KUKA KRL program: Jacob_final_print.src

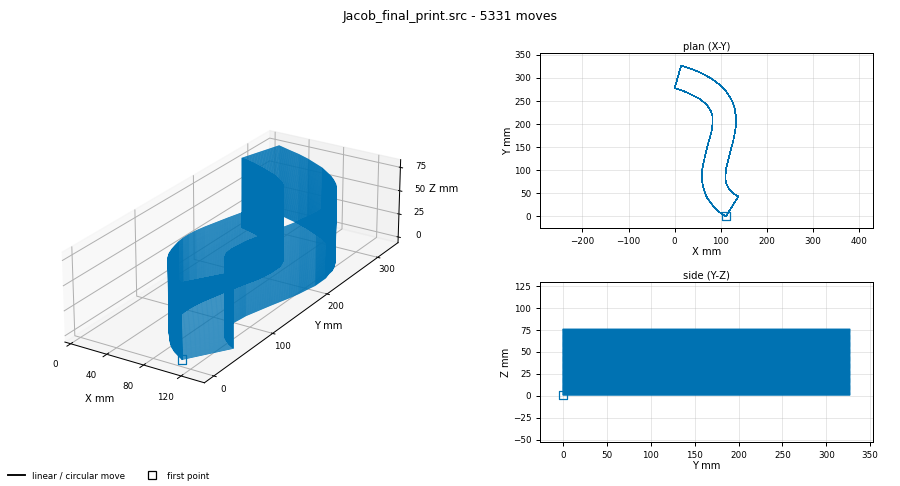
[picture p0: tool path of Jacob_final_print.src, 5331 of 5334 moves have a stored position in this frame; points joined in program order, loops and branches not executed]
&ACCESS RVP
&REL 25
DEF Jacob_final_print()

;FOLD INI
  ;FOLD BASISTECH INI
    GLOBAL INTERRUPT DECL 3 WHEN $STOPMESS==TRUE DO IR_STOPM ( )
    INTERRUPT ON 3
    BAS (#INITMOV,0 )
  ;ENDFOLD (BASISTECH INI)
  ;FOLD USER INI
    ;Make your modifications here

  ;ENDFOLD (USER INI)
;ENDFOLD (INI)

;FOLD PTP HOME  Vel= 100 % DEFAULT;%{PE}%R 5.4.37,%MKUKATPBASIS,%CMOVE,%VPTP,%P 1:PTP, 2:HOME, 3:, 5:100, 7:DEFAULT
$BWDSTART=FALSE
PDAT_ACT=PDEFAULT
FDAT_ACT=FHOME
BAS(#PTP_PARAMS,100)
$H_POS=XHOME
PTP XHOME
;ENDFOLD

$VEL_AXIS[1]=20
$VEL_AXIS[2]=20
$VEL_AXIS[3]=20
$VEL_AXIS[4]=20
$VEL_AXIS[5]=20
$VEL_AXIS[6]=20

$vel.cp= 0.30
$apo.cvel= 95

PTP {A1 0, A2 -90, A3 90, A4 0, A5 0, A6 0}

PTP {Z 450, S 110}

LIN {X 111, Y 0, Z 1} c_vel
$OUT[4] = TRUE
LIN {X 111, Y 0, Z 1} c_vel
LIN {X 106, Y 3, Z 1} c_vel
LIN {X 97, Y 9, Z 1} c_vel
LIN {X 89, Y 16, Z 1} c_vel
LIN {X 83, Y 23, Z 1} c_vel
LIN {X 77, Y 31, Z 1} c_vel
LIN {X 71, Y 39, Z 1} c_vel
LIN {X 67, Y 47, Z 1} c_vel
LIN {X 64, Y 56, Z 1} c_vel
LIN {X 62, Y 64, Z 1} c_vel
LIN {X 60, Y 73, Z 1} c_vel
LIN {X 59, Y 82, Z 1} c_vel
LIN {X 59, Y 82, Z 1} c_vel
LIN {X 59, Y 92, Z 1} c_vel
LIN {X 60, Y 103, Z 1} c_vel
LIN {X 62, Y 114, Z 1} c_vel
LIN {X 65, Y 127, Z 1} c_vel
LIN {X 69, Y 144, Z 1} c_vel
LIN {X 74, Y 163, Z 1} c_vel
LIN {X 79, Y 180, Z 1} c_vel
LIN {X 81, Y 191, Z 1} c_vel
LIN {X 82, Y 201, Z 1} c_vel
LIN {X 82, Y 209, Z 1} c_vel
LIN {X 82, Y 217, Z 1} c_vel
LIN {X 80, Y 223, Z 1} c_vel
LIN {X 78, Y 229, Z 1} c_vel
LIN {X 75, Y 234, Z 1} c_vel
LIN {X 71, Y 240, Z 1} c_vel
LIN {X 66, Y 245, Z 1} c_vel
LIN {X 60, Y 250, Z 1} c_vel
LIN {X 52, Y 256, Z 1} c_vel
LIN {X 42, Y 261, Z 1} c_vel
LIN {X 30, Y 267, Z 1} c_vel
LIN {X 16, Y 273, Z 1} c_vel
LIN {X 0, Y 278, Z 1} c_vel
LIN {X 14, Y 327, Z 1} c_vel
LIN {X 28, Y 322, Z 1} c_vel
LIN {X 43, Y 317, Z 1} c_vel
LIN {X 57, Y 311, Z 1} c_vel
LIN {X 70, Y 304, Z 1} c_vel
LIN {X 81, Y 298, Z 1} c_vel
LIN {X 90, Y 291, Z 1} c_vel
LIN {X 99, Y 284, Z 1} c_vel
LIN {X 106, Y 277, Z 1} c_vel
LIN {X 113, Y 269, Z 1} c_vel
LIN {X 118, Y 261, Z 1} c_vel
LIN {X 123, Y 253, Z 1} c_vel
LIN {X 127, Y 244, Z 1} c_vel
LIN {X 130, Y 235, Z 1} c_vel
LIN {X 131, Y 226, Z 1} c_vel
LIN {X 133, Y 217, Z 1} c_vel
LIN {X 133, Y 207, Z 1} c_vel
LIN {X 133, Y 197, Z 1} c_vel
LIN {X 131, Y 186, Z 1} c_vel
LIN {X 129, Y 173, Z 1} c_vel
LIN {X 126, Y 160, Z 1} c_vel
LIN {X 120, Y 138, Z 1} c_vel
LIN {X 115, Y 118, Z 1} c_vel
LIN {X 112, Y 106, Z 1} c_vel
LIN {X 111, Y 96, Z 1} c_vel
LIN {X 110, Y 88, Z 1} c_vel
LIN {X 110, Y 81, Z 1} c_vel
LIN {X 111, Y 74, Z 1} c_vel
LIN {X 113, Y 69, Z 1} c_vel
LIN {X 116, Y 63, Z 1} c_vel
LIN {X 119, Y 58, Z 1} c_vel
LIN {X 124, Y 53, Z 1} c_vel
LIN {X 130, Y 48, Z 1} c_vel
LIN {X 138, Y 43, Z 1} c_vel
LIN {X 111, Y 0, Z 1} c_vel
$OUT[4] = FALSE
WAIT SEC 10.0
LIN {X 111, Y 0, Z 2} c_vel
$OUT[4] = TRUE
LIN {X 111, Y 0, Z 2} c_vel
LIN {X 106, Y 3, Z 2} c_vel
LIN {X 97, Y 9, Z 2} c_vel
LIN {X 89, Y 16, Z 2} c_vel
LIN {X 83, Y 23, Z 2} c_vel
LIN {X 77, Y 31, Z 2} c_vel
LIN {X 71, Y 39, Z 2} c_vel
LIN {X 67, Y 47, Z 2} c_vel
LIN {X 64, Y 56, Z 2} c_vel
LIN {X 62, Y 64, Z 2} c_vel
LIN {X 60, Y 73, Z 2} c_vel
LIN {X 59, Y 82, Z 2} c_vel
LIN {X 59, Y 83, Z 2} c_vel
LIN {X 59, Y 92, Z 2} c_vel
LIN {X 60, Y 103, Z 2} c_vel
LIN {X 62, Y 114, Z 2} c_vel
LIN {X 65, Y 127, Z 2} c_vel
LIN {X 69, Y 144, Z 2} c_vel
LIN {X 74, Y 163, Z 2} c_vel
LIN {X 79, Y 180, Z 2} c_vel
LIN {X 81, Y 191, Z 2} c_vel
LIN {X 82, Y 201, Z 2} c_vel
LIN {X 82, Y 209, Z 2} c_vel
LIN {X 82, Y 217, Z 2} c_vel
LIN {X 80, Y 223, Z 2} c_vel
LIN {X 78, Y 229, Z 2} c_vel
LIN {X 75, Y 234, Z 2} c_vel
LIN {X 71, Y 240, Z 2} c_vel
LIN {X 66, Y 245, Z 2} c_vel
LIN {X 60, Y 250, Z 2} c_vel
LIN {X 52, Y 256, Z 2} c_vel
LIN {X 42, Y 261, Z 2} c_vel
LIN {X 30, Y 267, Z 2} c_vel
LIN {X 16, Y 273, Z 2} c_vel
LIN {X 0, Y 278, Z 2} c_vel
LIN {X 14, Y 327, Z 2} c_vel
LIN {X 28, Y 322, Z 2} c_vel
LIN {X 43, Y 317, Z 2} c_vel
LIN {X 57, Y 311, Z 2} c_vel
LIN {X 70, Y 304, Z 2} c_vel
LIN {X 81, Y 298, Z 2} c_vel
LIN {X 90, Y 291, Z 2} c_vel
LIN {X 99, Y 284, Z 2} c_vel
LIN {X 106, Y 277, Z 2} c_vel
LIN {X 113, Y 269, Z 2} c_vel
LIN {X 118, Y 261, Z 2} c_vel
LIN {X 123, Y 253, Z 2} c_vel
LIN {X 127, Y 244, Z 2} c_vel
LIN {X 130, Y 235, Z 2} c_vel
LIN {X 131, Y 226, Z 2} c_vel
LIN {X 133, Y 217, Z 2} c_vel
LIN {X 133, Y 207, Z 2} c_vel
LIN {X 133, Y 197, Z 2} c_vel
LIN {X 131, Y 186, Z 2} c_vel
LIN {X 129, Y 173, Z 2} c_vel
LIN {X 126, Y 160, Z 2} c_vel
LIN {X 120, Y 138, Z 2} c_vel
LIN {X 115, Y 118, Z 2} c_vel
LIN {X 112, Y 106, Z 2} c_vel
LIN {X 111, Y 96, Z 2} c_vel
LIN {X 110, Y 88, Z 2} c_vel
LIN {X 110, Y 81, Z 2} c_vel
LIN {X 111, Y 74, Z 2} c_vel
LIN {X 113, Y 69, Z 2} c_vel
LIN {X 116, Y 63, Z 2} c_vel
LIN {X 119, Y 58, Z 2} c_vel
LIN {X 124, Y 53, Z 2} c_vel
LIN {X 130, Y 48, Z 2} c_vel
LIN {X 138, Y 43, Z 2} c_vel
LIN {X 111, Y 0, Z 2} c_vel
$OUT[4] = FALSE
WAIT SEC 10.0
LIN {X 111, Y 0, Z 3} c_vel
$OUT[4] = TRUE
LIN {X 111, Y 0, Z 3} c_vel
LIN {X 106, Y 3, Z 3} c_vel
LIN {X 97, Y 9, Z 3} c_vel
LIN {X 89, Y 16, Z 3} c_vel
LIN {X 83, Y 23, Z 3} c_vel
LIN {X 77, Y 31, Z 3} c_vel
LIN {X 71, Y 39, Z 3} c_vel
LIN {X 67, Y 47, Z 3} c_vel
LIN {X 64, Y 56, Z 3} c_vel
LIN {X 62, Y 64, Z 3} c_vel
LIN {X 60, Y 73, Z 3} c_vel
LIN {X 59, Y 82, Z 3} c_vel
LIN {X 59, Y 83, Z 3} c_vel
LIN {X 59, Y 92, Z 3} c_vel
LIN {X 60, Y 103, Z 3} c_vel
LIN {X 62, Y 114, Z 3} c_vel
LIN {X 65, Y 127, Z 3} c_vel
LIN {X 69, Y 144, Z 3} c_vel
LIN {X 74, Y 163, Z 3} c_vel
LIN {X 79, Y 180, Z 3} c_vel
LIN {X 81, Y 191, Z 3} c_vel
LIN {X 82, Y 201, Z 3} c_vel
LIN {X 82, Y 209, Z 3} c_vel
LIN {X 82, Y 217, Z 3} c_vel
LIN {X 80, Y 223, Z 3} c_vel
LIN {X 78, Y 229, Z 3} c_vel
LIN {X 75, Y 234, Z 3} c_vel
LIN {X 71, Y 240, Z 3} c_vel
LIN {X 66, Y 245, Z 3} c_vel
LIN {X 60, Y 250, Z 3} c_vel
LIN {X 52, Y 256, Z 3} c_vel
LIN {X 42, Y 261, Z 3} c_vel
LIN {X 30, Y 267, Z 3} c_vel
LIN {X 16, Y 273, Z 3} c_vel
LIN {X 0, Y 278, Z 3} c_vel
LIN {X 14, Y 327, Z 3} c_vel
LIN {X 28, Y 322, Z 3} c_vel
LIN {X 43, Y 317, Z 3} c_vel
LIN {X 57, Y 311, Z 3} c_vel
LIN {X 70, Y 304, Z 3} c_vel
LIN {X 81, Y 298, Z 3} c_vel
LIN {X 90, Y 291, Z 3} c_vel
LIN {X 99, Y 284, Z 3} c_vel
LIN {X 106, Y 277, Z 3} c_vel
LIN {X 113, Y 269, Z 3} c_vel
LIN {X 118, Y 261, Z 3} c_vel
LIN {X 123, Y 253, Z 3} c_vel
LIN {X 127, Y 244, Z 3} c_vel
LIN {X 130, Y 235, Z 3} c_vel
LIN {X 131, Y 226, Z 3} c_vel
LIN {X 133, Y 217, Z 3} c_vel
LIN {X 133, Y 207, Z 3} c_vel
LIN {X 133, Y 197, Z 3} c_vel
LIN {X 131, Y 186, Z 3} c_vel
LIN {X 129, Y 173, Z 3} c_vel
LIN {X 126, Y 160, Z 3} c_vel
LIN {X 120, Y 138, Z 3} c_vel
LIN {X 115, Y 118, Z 3} c_vel
LIN {X 112, Y 106, Z 3} c_vel
LIN {X 111, Y 96, Z 3} c_vel
LIN {X 110, Y 88, Z 3} c_vel
LIN {X 110, Y 81, Z 3} c_vel
LIN {X 111, Y 74, Z 3} c_vel
LIN {X 113, Y 69, Z 3} c_vel
LIN {X 116, Y 63, Z 3} c_vel
LIN {X 119, Y 58, Z 3} c_vel
LIN {X 124, Y 53, Z 3} c_vel
LIN {X 130, Y 48, Z 3} c_vel
LIN {X 138, Y 43, Z 3} c_vel
LIN {X 111, Y 0, Z 3} c_vel
$OUT[4] = FALSE
WAIT SEC 10.0
LIN {X 111, Y 0, Z 4} c_vel
$OUT[4] = TRUE
LIN {X 111, Y 0, Z 4} c_vel
LIN {X 106, Y 3, Z 4} c_vel
LIN {X 97, Y 9, Z 4} c_vel
LIN {X 89, Y 16, Z 4} c_vel
LIN {X 83, Y 23, Z 4} c_vel
LIN {X 77, Y 31, Z 4} c_vel
LIN {X 71, Y 39, Z 4} c_vel
LIN {X 67, Y 47, Z 4} c_vel
LIN {X 64, Y 56, Z 4} c_vel
LIN {X 62, Y 64, Z 4} c_vel
LIN {X 60, Y 73, Z 4} c_vel
LIN {X 59, Y 82, Z 4} c_vel
LIN {X 59, Y 83, Z 4} c_vel
LIN {X 59, Y 92, Z 4} c_vel
LIN {X 60, Y 103, Z 4} c_vel
LIN {X 62, Y 114, Z 4} c_vel
LIN {X 65, Y 127, Z 4} c_vel
LIN {X 69, Y 144, Z 4} c_vel
LIN {X 74, Y 163, Z 4} c_vel
LIN {X 79, Y 180, Z 4} c_vel
LIN {X 81, Y 191, Z 4} c_vel
LIN {X 82, Y 201, Z 4} c_vel
LIN {X 82, Y 209, Z 4} c_vel
LIN {X 82, Y 217, Z 4} c_vel
LIN {X 80, Y 223, Z 4} c_vel
LIN {X 78, Y 229, Z 4} c_vel
LIN {X 75, Y 234, Z 4} c_vel
LIN {X 71, Y 240, Z 4} c_vel
LIN {X 66, Y 245, Z 4} c_vel
LIN {X 60, Y 250, Z 4} c_vel
LIN {X 52, Y 256, Z 4} c_vel
LIN {X 42, Y 261, Z 4} c_vel
LIN {X 30, Y 267, Z 4} c_vel
LIN {X 16, Y 273, Z 4} c_vel
LIN {X 0, Y 278, Z 4} c_vel
LIN {X 14, Y 327, Z 4} c_vel
LIN {X 28, Y 322, Z 4} c_vel
LIN {X 43, Y 317, Z 4} c_vel
LIN {X 57, Y 311, Z 4} c_vel
LIN {X 70, Y 304, Z 4} c_vel
LIN {X 81, Y 298, Z 4} c_vel
LIN {X 90, Y 291, Z 4} c_vel
LIN {X 99, Y 284, Z 4} c_vel
LIN {X 106, Y 277, Z 4} c_vel
LIN {X 113, Y 269, Z 4} c_vel
LIN {X 118, Y 261, Z 4} c_vel
LIN {X 123, Y 253, Z 4} c_vel
LIN {X 127, Y 244, Z 4} c_vel
LIN {X 130, Y 235, Z 4} c_vel
LIN {X 131, Y 226, Z 4} c_vel
LIN {X 133, Y 217, Z 4} c_vel
LIN {X 133, Y 207, Z 4} c_vel
LIN {X 133, Y 197, Z 4} c_vel
LIN {X 131, Y 186, Z 4} c_vel
LIN {X 129, Y 173, Z 4} c_vel
LIN {X 126, Y 160, Z 4} c_vel
LIN {X 120, Y 138, Z 4} c_vel
LIN {X 115, Y 118, Z 4} c_vel
LIN {X 112, Y 106, Z 4} c_vel
LIN {X 111, Y 96, Z 4} c_vel
LIN {X 110, Y 88, Z 4} c_vel
LIN {X 110, Y 81, Z 4} c_vel
LIN {X 111, Y 74, Z 4} c_vel
LIN {X 113, Y 69, Z 4} c_vel
LIN {X 116, Y 63, Z 4} c_vel
LIN {X 119, Y 58, Z 4} c_vel
LIN {X 124, Y 53, Z 4} c_vel
LIN {X 130, Y 48, Z 4} c_vel
LIN {X 138, Y 43, Z 4} c_vel
LIN {X 111, Y 0, Z 4} c_vel
$OUT[4] = FALSE
WAIT SEC 10.0
LIN {X 111, Y 0, Z 5} c_vel
$OUT[4] = TRUE
LIN {X 111, Y 0, Z 5} c_vel
LIN {X 106, Y 3, Z 5} c_vel
LIN {X 97, Y 9, Z 5} c_vel
LIN {X 89, Y 16, Z 5} c_vel
LIN {X 83, Y 23, Z 5} c_vel
LIN {X 77, Y 31, Z 5} c_vel
LIN {X 71, Y 39, Z 5} c_vel
LIN {X 67, Y 47, Z 5} c_vel
LIN {X 64, Y 56, Z 5} c_vel
LIN {X 62, Y 64, Z 5} c_vel
LIN {X 60, Y 73, Z 5} c_vel
LIN {X 59, Y 82, Z 5} c_vel
LIN {X 59, Y 83, Z 5} c_vel
LIN {X 59, Y 92, Z 5} c_vel
LIN {X 60, Y 103, Z 5} c_vel
LIN {X 62, Y 114, Z 5} c_vel
LIN {X 65, Y 127, Z 5} c_vel
LIN {X 69, Y 144, Z 5} c_vel
LIN {X 74, Y 163, Z 5} c_vel
LIN {X 79, Y 180, Z 5} c_vel
LIN {X 81, Y 191, Z 5} c_vel
LIN {X 82, Y 201, Z 5} c_vel
LIN {X 82, Y 209, Z 5} c_vel
LIN {X 82, Y 217, Z 5} c_vel
LIN {X 80, Y 223, Z 5} c_vel
LIN {X 78, Y 229, Z 5} c_vel
LIN {X 75, Y 234, Z 5} c_vel
LIN {X 71, Y 240, Z 5} c_vel
LIN {X 66, Y 245, Z 5} c_vel
LIN {X 60, Y 250, Z 5} c_vel
LIN {X 52, Y 256, Z 5} c_vel
LIN {X 42, Y 261, Z 5} c_vel
LIN {X 30, Y 267, Z 5} c_vel
LIN {X 16, Y 273, Z 5} c_vel
LIN {X 0, Y 278, Z 5} c_vel
LIN {X 14, Y 327, Z 5} c_vel
LIN {X 28, Y 322, Z 5} c_vel
LIN {X 43, Y 317, Z 5} c_vel
LIN {X 57, Y 311, Z 5} c_vel
LIN {X 70, Y 304, Z 5} c_vel
LIN {X 81, Y 298, Z 5} c_vel
LIN {X 90, Y 291, Z 5} c_vel
LIN {X 99, Y 284, Z 5} c_vel
LIN {X 106, Y 277, Z 5} c_vel
LIN {X 113, Y 269, Z 5} c_vel
LIN {X 118, Y 261, Z 5} c_vel
LIN {X 123, Y 253, Z 5} c_vel
LIN {X 127, Y 244, Z 5} c_vel
LIN {X 130, Y 235, Z 5} c_vel
LIN {X 131, Y 226, Z 5} c_vel
LIN {X 133, Y 217, Z 5} c_vel
LIN {X 133, Y 207, Z 5} c_vel
LIN {X 133, Y 197, Z 5} c_vel
LIN {X 131, Y 186, Z 5} c_vel
LIN {X 129, Y 173, Z 5} c_vel
LIN {X 126, Y 160, Z 5} c_vel
LIN {X 120, Y 138, Z 5} c_vel
LIN {X 115, Y 118, Z 5} c_vel
LIN {X 112, Y 106, Z 5} c_vel
LIN {X 111, Y 96, Z 5} c_vel
LIN {X 110, Y 88, Z 5} c_vel
LIN {X 110, Y 81, Z 5} c_vel
LIN {X 111, Y 74, Z 5} c_vel
LIN {X 113, Y 69, Z 5} c_vel
LIN {X 116, Y 63, Z 5} c_vel
LIN {X 119, Y 58, Z 5} c_vel
LIN {X 124, Y 53, Z 5} c_vel
LIN {X 130, Y 48, Z 5} c_vel
LIN {X 138, Y 43, Z 5} c_vel
LIN {X 111, Y 0, Z 5} c_vel
$OUT[4] = FALSE
WAIT SEC 10.0
LIN {X 111, Y 0, Z 6} c_vel
$OUT[4] = TRUE
LIN {X 111, Y 0, Z 6} c_vel
LIN {X 106, Y 3, Z 6} c_vel
LIN {X 97, Y 9, Z 6} c_vel
LIN {X 89, Y 16, Z 6} c_vel
LIN {X 83, Y 23, Z 6} c_vel
LIN {X 77, Y 31, Z 6} c_vel
LIN {X 71, Y 39, Z 6} c_vel
LIN {X 67, Y 47, Z 6} c_vel
LIN {X 64, Y 56, Z 6} c_vel
LIN {X 62, Y 64, Z 6} c_vel
LIN {X 60, Y 73, Z 6} c_vel
LIN {X 59, Y 82, Z 6} c_vel
LIN {X 59, Y 83, Z 6} c_vel
LIN {X 59, Y 92, Z 6} c_vel
LIN {X 60, Y 103, Z 6} c_vel
LIN {X 62, Y 114, Z 6} c_vel
LIN {X 65, Y 127, Z 6} c_vel
LIN {X 69, Y 144, Z 6} c_vel
LIN {X 74, Y 163, Z 6} c_vel
LIN {X 79, Y 180, Z 6} c_vel
LIN {X 81, Y 191, Z 6} c_vel
LIN {X 82, Y 201, Z 6} c_vel
LIN {X 82, Y 209, Z 6} c_vel
LIN {X 82, Y 217, Z 6} c_vel
LIN {X 80, Y 223, Z 6} c_vel
LIN {X 78, Y 229, Z 6} c_vel
LIN {X 75, Y 234, Z 6} c_vel
LIN {X 71, Y 240, Z 6} c_vel
LIN {X 66, Y 245, Z 6} c_vel
LIN {X 60, Y 250, Z 6} c_vel
LIN {X 52, Y 256, Z 6} c_vel
LIN {X 42, Y 261, Z 6} c_vel
LIN {X 30, Y 267, Z 6} c_vel
LIN {X 16, Y 273, Z 6} c_vel
LIN {X 0, Y 278, Z 6} c_vel
LIN {X 14, Y 327, Z 6} c_vel
LIN {X 28, Y 322, Z 6} c_vel
LIN {X 43, Y 317, Z 6} c_vel
LIN {X 57, Y 311, Z 6} c_vel
LIN {X 70, Y 304, Z 6} c_vel
LIN {X 81, Y 298, Z 6} c_vel
LIN {X 90, Y 291, Z 6} c_vel
LIN {X 99, Y 284, Z 6} c_vel
LIN {X 106, Y 277, Z 6} c_vel
LIN {X 113, Y 269, Z 6} c_vel
LIN {X 118, Y 261, Z 6} c_vel
LIN {X 123, Y 253, Z 6} c_vel
LIN {X 127, Y 244, Z 6} c_vel
LIN {X 130, Y 235, Z 6} c_vel
LIN {X 131, Y 226, Z 6} c_vel
LIN {X 133, Y 217, Z 6} c_vel
LIN {X 133, Y 207, Z 6} c_vel
LIN {X 133, Y 197, Z 6} c_vel
LIN {X 131, Y 186, Z 6} c_vel
LIN {X 129, Y 173, Z 6} c_vel
LIN {X 126, Y 160, Z 6} c_vel
LIN {X 120, Y 138, Z 6} c_vel
LIN {X 115, Y 118, Z 6} c_vel
LIN {X 112, Y 106, Z 6} c_vel
LIN {X 111, Y 96, Z 6} c_vel
LIN {X 110, Y 88, Z 6} c_vel
LIN {X 110, Y 81, Z 6} c_vel
LIN {X 111, Y 74, Z 6} c_vel
LIN {X 113, Y 69, Z 6} c_vel
LIN {X 116, Y 63, Z 6} c_vel
LIN {X 119, Y 58, Z 6} c_vel
LIN {X 124, Y 53, Z 6} c_vel
LIN {X 130, Y 48, Z 6} c_vel
LIN {X 138, Y 43, Z 6} c_vel
LIN {X 111, Y 0, Z 6} c_vel
$OUT[4] = FALSE
WAIT SEC 10.0
LIN {X 111, Y 0, Z 7} c_vel
$OUT[4] = TRUE
LIN {X 111, Y 0, Z 7} c_vel
LIN {X 106, Y 3, Z 7} c_vel
LIN {X 97, Y 9, Z 7} c_vel
LIN {X 89, Y 16, Z 7} c_vel
LIN {X 83, Y 23, Z 7} c_vel
LIN {X 77, Y 31, Z 7} c_vel
LIN {X 71, Y 39, Z 7} c_vel
LIN {X 67, Y 47, Z 7} c_vel
LIN {X 64, Y 56, Z 7} c_vel
LIN {X 62, Y 64, Z 7} c_vel
LIN {X 60, Y 73, Z 7} c_vel
LIN {X 59, Y 82, Z 7} c_vel
LIN {X 59, Y 92, Z 7} c_vel
LIN {X 60, Y 103, Z 7} c_vel
LIN {X 62, Y 114, Z 7} c_vel
LIN {X 65, Y 127, Z 7} c_vel
LIN {X 69, Y 144, Z 7} c_vel
LIN {X 74, Y 163, Z 7} c_vel
LIN {X 79, Y 180, Z 7} c_vel
LIN {X 81, Y 191, Z 7} c_vel
LIN {X 82, Y 201, Z 7} c_vel
LIN {X 82, Y 209, Z 7} c_vel
LIN {X 82, Y 217, Z 7} c_vel
LIN {X 80, Y 223, Z 7} c_vel
LIN {X 78, Y 229, Z 7} c_vel
LIN {X 75, Y 234, Z 7} c_vel
LIN {X 71, Y 240, Z 7} c_vel
LIN {X 66, Y 245, Z 7} c_vel
LIN {X 60, Y 250, Z 7} c_vel
LIN {X 52, Y 256, Z 7} c_vel
LIN {X 42, Y 261, Z 7} c_vel
LIN {X 30, Y 267, Z 7} c_vel
LIN {X 16, Y 273, Z 7} c_vel
LIN {X 0, Y 278, Z 7} c_vel
LIN {X 14, Y 327, Z 7} c_vel
LIN {X 28, Y 322, Z 7} c_vel
LIN {X 43, Y 317, Z 7} c_vel
LIN {X 57, Y 311, Z 7} c_vel
LIN {X 70, Y 304, Z 7} c_vel
LIN {X 81, Y 298, Z 7} c_vel
LIN {X 90, Y 291, Z 7} c_vel
LIN {X 99, Y 284, Z 7} c_vel
LIN {X 106, Y 277, Z 7} c_vel
LIN {X 113, Y 269, Z 7} c_vel
LIN {X 118, Y 261, Z 7} c_vel
LIN {X 123, Y 253, Z 7} c_vel
LIN {X 127, Y 244, Z 7} c_vel
LIN {X 130, Y 235, Z 7} c_vel
LIN {X 131, Y 226, Z 7} c_vel
LIN {X 133, Y 217, Z 7} c_vel
LIN {X 133, Y 207, Z 7} c_vel
LIN {X 133, Y 197, Z 7} c_vel
LIN {X 131, Y 186, Z 7} c_vel
LIN {X 129, Y 173, Z 7} c_vel
LIN {X 126, Y 160, Z 7} c_vel
LIN {X 120, Y 138, Z 7} c_vel
LIN {X 115, Y 118, Z 7} c_vel
LIN {X 112, Y 106, Z 7} c_vel
LIN {X 111, Y 96, Z 7} c_vel
LIN {X 110, Y 88, Z 7} c_vel
LIN {X 110, Y 81, Z 7} c_vel
LIN {X 111, Y 74, Z 7} c_vel
LIN {X 113, Y 69, Z 7} c_vel
LIN {X 116, Y 63, Z 7} c_vel
LIN {X 119, Y 58, Z 7} c_vel
LIN {X 124, Y 53, Z 7} c_vel
LIN {X 130, Y 48, Z 7} c_vel
LIN {X 138, Y 43, Z 7} c_vel
LIN {X 111, Y 0, Z 7} c_vel
$OUT[4] = FALSE
WAIT SEC 10.0
LIN {X 111, Y 0, Z 8} c_vel
$OUT[4] = TRUE
LIN {X 111, Y 0, Z 8} c_vel
LIN {X 106, Y 3, Z 8} c_vel
LIN {X 97, Y 9, Z 8} c_vel
LIN {X 89, Y 16, Z 8} c_vel
LIN {X 83, Y 23, Z 8} c_vel
LIN {X 77, Y 31, Z 8} c_vel
LIN {X 71, Y 39, Z 8} c_vel
LIN {X 67, Y 47, Z 8} c_vel
LIN {X 64, Y 56, Z 8} c_vel
LIN {X 62, Y 64, Z 8} c_vel
LIN {X 60, Y 73, Z 8} c_vel
LIN {X 59, Y 82, Z 8} c_vel
LIN {X 59, Y 92, Z 8} c_vel
LIN {X 60, Y 103, Z 8} c_vel
LIN {X 62, Y 114, Z 8} c_vel
LIN {X 65, Y 127, Z 8} c_vel
LIN {X 69, Y 144, Z 8} c_vel
LIN {X 74, Y 163, Z 8} c_vel
LIN {X 79, Y 180, Z 8} c_vel
LIN {X 81, Y 191, Z 8} c_vel
LIN {X 82, Y 201, Z 8} c_vel
LIN {X 82, Y 209, Z 8} c_vel
LIN {X 82, Y 217, Z 8} c_vel
LIN {X 80, Y 223, Z 8} c_vel
LIN {X 78, Y 229, Z 8} c_vel
LIN {X 75, Y 234, Z 8} c_vel
LIN {X 71, Y 240, Z 8} c_vel
LIN {X 66, Y 245, Z 8} c_vel
LIN {X 60, Y 250, Z 8} c_vel
LIN {X 52, Y 256, Z 8} c_vel
LIN {X 42, Y 261, Z 8} c_vel
LIN {X 30, Y 267, Z 8} c_vel
LIN {X 16, Y 273, Z 8} c_vel
LIN {X 0, Y 278, Z 8} c_vel
LIN {X 14, Y 327, Z 8} c_vel
LIN {X 28, Y 322, Z 8} c_vel
LIN {X 43, Y 317, Z 8} c_vel
LIN {X 57, Y 311, Z 8} c_vel
LIN {X 70, Y 304, Z 8} c_vel
LIN {X 81, Y 298, Z 8} c_vel
LIN {X 90, Y 291, Z 8} c_vel
LIN {X 99, Y 284, Z 8} c_vel
LIN {X 106, Y 277, Z 8} c_vel
LIN {X 113, Y 269, Z 8} c_vel
LIN {X 118, Y 261, Z 8} c_vel
LIN {X 123, Y 253, Z 8} c_vel
LIN {X 127, Y 244, Z 8} c_vel
LIN {X 130, Y 235, Z 8} c_vel
LIN {X 131, Y 226, Z 8} c_vel
LIN {X 133, Y 217, Z 8} c_vel
LIN {X 133, Y 207, Z 8} c_vel
LIN {X 133, Y 197, Z 8} c_vel
LIN {X 131, Y 186, Z 8} c_vel
LIN {X 129, Y 173, Z 8} c_vel
LIN {X 126, Y 160, Z 8} c_vel
LIN {X 120, Y 138, Z 8} c_vel
LIN {X 115, Y 118, Z 8} c_vel
LIN {X 112, Y 106, Z 8} c_vel
LIN {X 111, Y 96, Z 8} c_vel
LIN {X 110, Y 88, Z 8} c_vel
LIN {X 110, Y 81, Z 8} c_vel
LIN {X 111, Y 74, Z 8} c_vel
LIN {X 113, Y 69, Z 8} c_vel
LIN {X 116, Y 63, Z 8} c_vel
LIN {X 119, Y 58, Z 8} c_vel
LIN {X 124, Y 53, Z 8} c_vel
LIN {X 130, Y 48, Z 8} c_vel
LIN {X 138, Y 43, Z 8} c_vel
LIN {X 111, Y 0, Z 8} c_vel
$OUT[4] = FALSE
WAIT SEC 10.0
LIN {X 111, Y 0, Z 9} c_vel
$OUT[4] = TRUE
LIN {X 111, Y 0, Z 9} c_vel
LIN {X 106, Y 3, Z 9} c_vel
LIN {X 97, Y 9, Z 9} c_vel
LIN {X 89, Y 16, Z 9} c_vel
LIN {X 83, Y 23, Z 9} c_vel
LIN {X 77, Y 31, Z 9} c_vel
LIN {X 71, Y 39, Z 9} c_vel
LIN {X 67, Y 47, Z 9} c_vel
LIN {X 64, Y 56, Z 9} c_vel
LIN {X 62, Y 64, Z 9} c_vel
LIN {X 60, Y 73, Z 9} c_vel
LIN {X 59, Y 82, Z 9} c_vel
LIN {X 59, Y 92, Z 9} c_vel
LIN {X 60, Y 103, Z 9} c_vel
LIN {X 62, Y 114, Z 9} c_vel
LIN {X 65, Y 127, Z 9} c_vel
LIN {X 69, Y 144, Z 9} c_vel
LIN {X 74, Y 163, Z 9} c_vel
LIN {X 79, Y 180, Z 9} c_vel
LIN {X 81, Y 191, Z 9} c_vel
LIN {X 82, Y 201, Z 9} c_vel
LIN {X 82, Y 209, Z 9} c_vel
LIN {X 82, Y 217, Z 9} c_vel
LIN {X 80, Y 223, Z 9} c_vel
LIN {X 78, Y 229, Z 9} c_vel
LIN {X 75, Y 234, Z 9} c_vel
LIN {X 71, Y 240, Z 9} c_vel
LIN {X 66, Y 245, Z 9} c_vel
LIN {X 60, Y 250, Z 9} c_vel
LIN {X 52, Y 256, Z 9} c_vel
LIN {X 42, Y 261, Z 9} c_vel
LIN {X 30, Y 267, Z 9} c_vel
LIN {X 16, Y 273, Z 9} c_vel
LIN {X 0, Y 278, Z 9} c_vel
LIN {X 14, Y 327, Z 9} c_vel
LIN {X 28, Y 322, Z 9} c_vel
LIN {X 43, Y 317, Z 9} c_vel
LIN {X 57, Y 311, Z 9} c_vel
LIN {X 70, Y 304, Z 9} c_vel
LIN {X 81, Y 298, Z 9} c_vel
LIN {X 90, Y 291, Z 9} c_vel
LIN {X 99, Y 284, Z 9} c_vel
LIN {X 106, Y 277, Z 9} c_vel
LIN {X 113, Y 269, Z 9} c_vel
LIN {X 118, Y 261, Z 9} c_vel
LIN {X 123, Y 253, Z 9} c_vel
LIN {X 127, Y 244, Z 9} c_vel
LIN {X 130, Y 235, Z 9} c_vel
LIN {X 131, Y 226, Z 9} c_vel
LIN {X 133, Y 217, Z 9} c_vel
LIN {X 133, Y 207, Z 9} c_vel
LIN {X 133, Y 197, Z 9} c_vel
LIN {X 131, Y 186, Z 9} c_vel
LIN {X 129, Y 173, Z 9} c_vel
LIN {X 126, Y 160, Z 9} c_vel
LIN {X 120, Y 138, Z 9} c_vel
LIN {X 115, Y 118, Z 9} c_vel
LIN {X 112, Y 106, Z 9} c_vel
LIN {X 111, Y 96, Z 9} c_vel
LIN {X 110, Y 88, Z 9} c_vel
LIN {X 110, Y 81, Z 9} c_vel
LIN {X 111, Y 74, Z 9} c_vel
LIN {X 113, Y 69, Z 9} c_vel
LIN {X 116, Y 63, Z 9} c_vel
LIN {X 119, Y 58, Z 9} c_vel
LIN {X 124, Y 53, Z 9} c_vel
LIN {X 130, Y 48, Z 9} c_vel
LIN {X 138, Y 43, Z 9} c_vel
LIN {X 111, Y 0, Z 9} c_vel
$OUT[4] = FALSE
WAIT SEC 10.0
LIN {X 111, Y 0, Z 10} c_vel
$OUT[4] = TRUE
LIN {X 111, Y 0, Z 10} c_vel
LIN {X 106, Y 3, Z 10} c_vel
LIN {X 97, Y 9, Z 10} c_vel
LIN {X 89, Y 16, Z 10} c_vel
LIN {X 83, Y 23, Z 10} c_vel
LIN {X 77, Y 31, Z 10} c_vel
LIN {X 71, Y 39, Z 10} c_vel
LIN {X 67, Y 47, Z 10} c_vel
LIN {X 64, Y 56, Z 10} c_vel
LIN {X 62, Y 64, Z 10} c_vel
LIN {X 60, Y 73, Z 10} c_vel
LIN {X 59, Y 82, Z 10} c_vel
LIN {X 59, Y 92, Z 10} c_vel
LIN {X 60, Y 103, Z 10} c_vel
LIN {X 62, Y 114, Z 10} c_vel
LIN {X 65, Y 127, Z 10} c_vel
LIN {X 69, Y 144, Z 10} c_vel
LIN {X 74, Y 163, Z 10} c_vel
LIN {X 79, Y 180, Z 10} c_vel
LIN {X 81, Y 191, Z 10} c_vel
LIN {X 82, Y 201, Z 10} c_vel
LIN {X 82, Y 209, Z 10} c_vel
LIN {X 82, Y 217, Z 10} c_vel
LIN {X 80, Y 223, Z 10} c_vel
LIN {X 78, Y 229, Z 10} c_vel
LIN {X 75, Y 234, Z 10} c_vel
LIN {X 71, Y 240, Z 10} c_vel
LIN {X 66, Y 245, Z 10} c_vel
LIN {X 60, Y 250, Z 10} c_vel
LIN {X 52, Y 256, Z 10} c_vel
LIN {X 42, Y 261, Z 10} c_vel
LIN {X 30, Y 267, Z 10} c_vel
LIN {X 16, Y 273, Z 10} c_vel
LIN {X 0, Y 278, Z 10} c_vel
LIN {X 14, Y 327, Z 10} c_vel
LIN {X 28, Y 322, Z 10} c_vel
LIN {X 43, Y 317, Z 10} c_vel
LIN {X 57, Y 311, Z 10} c_vel
LIN {X 70, Y 304, Z 10} c_vel
LIN {X 81, Y 298, Z 10} c_vel
LIN {X 90, Y 291, Z 10} c_vel
LIN {X 99, Y 284, Z 10} c_vel
LIN {X 106, Y 277, Z 10} c_vel
LIN {X 113, Y 269, Z 10} c_vel
LIN {X 118, Y 261, Z 10} c_vel
LIN {X 123, Y 253, Z 10} c_vel
LIN {X 127, Y 244, Z 10} c_vel
LIN {X 130, Y 235, Z 10} c_vel
LIN {X 131, Y 226, Z 10} c_vel
LIN {X 133, Y 217, Z 10} c_vel
LIN {X 133, Y 207, Z 10} c_vel
LIN {X 133, Y 197, Z 10} c_vel
LIN {X 131, Y 186, Z 10} c_vel
LIN {X 129, Y 173, Z 10} c_vel
LIN {X 126, Y 160, Z 10} c_vel
LIN {X 120, Y 138, Z 10} c_vel
LIN {X 115, Y 118, Z 10} c_vel
LIN {X 112, Y 106, Z 10} c_vel
LIN {X 111, Y 96, Z 10} c_vel
LIN {X 110, Y 88, Z 10} c_vel
LIN {X 110, Y 81, Z 10} c_vel
LIN {X 111, Y 74, Z 10} c_vel
LIN {X 113, Y 69, Z 10} c_vel
LIN {X 116, Y 63, Z 10} c_vel
LIN {X 119, Y 58, Z 10} c_vel
LIN {X 124, Y 53, Z 10} c_vel
LIN {X 130, Y 48, Z 10} c_vel
LIN {X 138, Y 43, Z 10} c_vel
LIN {X 111, Y 0, Z 10} c_vel
$OUT[4] = FALSE
WAIT SEC 10.0
LIN {X 111, Y 0, Z 11} c_vel
$OUT[4] = TRUE
LIN {X 111, Y 0, Z 11} c_vel
LIN {X 106, Y 3, Z 11} c_vel
LIN {X 97, Y 9, Z 11} c_vel
LIN {X 89, Y 16, Z 11} c_vel
LIN {X 83, Y 23, Z 11} c_vel
LIN {X 77, Y 31, Z 11} c_vel
LIN {X 71, Y 39, Z 11} c_vel
LIN {X 67, Y 47, Z 11} c_vel
LIN {X 64, Y 56, Z 11} c_vel
LIN {X 62, Y 64, Z 11} c_vel
LIN {X 60, Y 73, Z 11} c_vel
LIN {X 59, Y 82, Z 11} c_vel
LIN {X 59, Y 92, Z 11} c_vel
LIN {X 60, Y 103, Z 11} c_vel
LIN {X 62, Y 114, Z 11} c_vel
LIN {X 65, Y 127, Z 11} c_vel
LIN {X 69, Y 144, Z 11} c_vel
LIN {X 74, Y 163, Z 11} c_vel
LIN {X 79, Y 180, Z 11} c_vel
LIN {X 81, Y 191, Z 11} c_vel
LIN {X 82, Y 201, Z 11} c_vel
LIN {X 82, Y 209, Z 11} c_vel
LIN {X 82, Y 217, Z 11} c_vel
LIN {X 80, Y 223, Z 11} c_vel
LIN {X 78, Y 229, Z 11} c_vel
LIN {X 75, Y 234, Z 11} c_vel
LIN {X 71, Y 240, Z 11} c_vel
LIN {X 66, Y 245, Z 11} c_vel
LIN {X 60, Y 250, Z 11} c_vel
LIN {X 52, Y 256, Z 11} c_vel
LIN {X 42, Y 261, Z 11} c_vel
LIN {X 30, Y 267, Z 11} c_vel
LIN {X 16, Y 273, Z 11} c_vel
LIN {X 0, Y 278, Z 11} c_vel
LIN {X 14, Y 327, Z 11} c_vel
LIN {X 28, Y 322, Z 11} c_vel
LIN {X 43, Y 317, Z 11} c_vel
LIN {X 57, Y 311, Z 11} c_vel
LIN {X 70, Y 304, Z 11} c_vel
LIN {X 81, Y 298, Z 11} c_vel
LIN {X 90, Y 291, Z 11} c_vel
LIN {X 99, Y 284, Z 11} c_vel
LIN {X 106, Y 277, Z 11} c_vel
LIN {X 113, Y 269, Z 11} c_vel
LIN {X 118, Y 261, Z 11} c_vel
LIN {X 123, Y 253, Z 11} c_vel
LIN {X 127, Y 244, Z 11} c_vel
LIN {X 130, Y 235, Z 11} c_vel
LIN {X 131, Y 226, Z 11} c_vel
LIN {X 133, Y 217, Z 11} c_vel
LIN {X 133, Y 207, Z 11} c_vel
LIN {X 133, Y 197, Z 11} c_vel
LIN {X 131, Y 186, Z 11} c_vel
LIN {X 129, Y 173, Z 11} c_vel
LIN {X 126, Y 160, Z 11} c_vel
LIN {X 120, Y 138, Z 11} c_vel
LIN {X 115, Y 118, Z 11} c_vel
LIN {X 112, Y 106, Z 11} c_vel
LIN {X 111, Y 96, Z 11} c_vel
LIN {X 110, Y 88, Z 11} c_vel
LIN {X 110, Y 81, Z 11} c_vel
LIN {X 111, Y 74, Z 11} c_vel
LIN {X 113, Y 69, Z 11} c_vel
LIN {X 116, Y 63, Z 11} c_vel
LIN {X 119, Y 58, Z 11} c_vel
LIN {X 124, Y 53, Z 11} c_vel
LIN {X 130, Y 48, Z 11} c_vel
LIN {X 138, Y 43, Z 11} c_vel
LIN {X 111, Y 0, Z 11} c_vel
$OUT[4] = FALSE
WAIT SEC 10.0
LIN {X 111, Y 0, Z 12} c_vel
$OUT[4] = TRUE
LIN {X 111, Y 0, Z 12} c_vel
LIN {X 106, Y 3, Z 12} c_vel
LIN {X 97, Y 9, Z 12} c_vel
LIN {X 89, Y 16, Z 12} c_vel
LIN {X 83, Y 23, Z 12} c_vel
LIN {X 77, Y 31, Z 12} c_vel
LIN {X 71, Y 39, Z 12} c_vel
LIN {X 67, Y 47, Z 12} c_vel
LIN {X 64, Y 56, Z 12} c_vel
LIN {X 62, Y 64, Z 12} c_vel
LIN {X 60, Y 73, Z 12} c_vel
LIN {X 59, Y 82, Z 12} c_vel
LIN {X 59, Y 92, Z 12} c_vel
LIN {X 60, Y 103, Z 12} c_vel
LIN {X 62, Y 114, Z 12} c_vel
LIN {X 65, Y 127, Z 12} c_vel
LIN {X 69, Y 144, Z 12} c_vel
LIN {X 74, Y 163, Z 12} c_vel
LIN {X 79, Y 180, Z 12} c_vel
LIN {X 81, Y 191, Z 12} c_vel
LIN {X 82, Y 201, Z 12} c_vel
LIN {X 82, Y 209, Z 12} c_vel
LIN {X 82, Y 217, Z 12} c_vel
LIN {X 80, Y 223, Z 12} c_vel
LIN {X 78, Y 229, Z 12} c_vel
LIN {X 75, Y 234, Z 12} c_vel
LIN {X 71, Y 240, Z 12} c_vel
LIN {X 66, Y 245, Z 12} c_vel
LIN {X 60, Y 250, Z 12} c_vel
LIN {X 52, Y 256, Z 12} c_vel
LIN {X 42, Y 261, Z 12} c_vel
LIN {X 30, Y 267, Z 12} c_vel
LIN {X 16, Y 273, Z 12} c_vel
LIN {X 0, Y 278, Z 12} c_vel
LIN {X 14, Y 327, Z 12} c_vel
LIN {X 28, Y 322, Z 12} c_vel
LIN {X 43, Y 317, Z 12} c_vel
LIN {X 57, Y 311, Z 12} c_vel
LIN {X 70, Y 304, Z 12} c_vel
LIN {X 81, Y 298, Z 12} c_vel
LIN {X 90, Y 291, Z 12} c_vel
LIN {X 99, Y 284, Z 12} c_vel
LIN {X 106, Y 277, Z 12} c_vel
LIN {X 113, Y 269, Z 12} c_vel
LIN {X 118, Y 261, Z 12} c_vel
LIN {X 123, Y 253, Z 12} c_vel
LIN {X 127, Y 244, Z 12} c_vel
LIN {X 130, Y 235, Z 12} c_vel
LIN {X 131, Y 226, Z 12} c_vel
LIN {X 133, Y 217, Z 12} c_vel
LIN {X 133, Y 207, Z 12} c_vel
LIN {X 133, Y 197, Z 12} c_vel
LIN {X 131, Y 186, Z 12} c_vel
LIN {X 129, Y 173, Z 12} c_vel
LIN {X 126, Y 160, Z 12} c_vel
LIN {X 120, Y 138, Z 12} c_vel
LIN {X 115, Y 118, Z 12} c_vel
LIN {X 112, Y 106, Z 12} c_vel
LIN {X 111, Y 96, Z 12} c_vel
LIN {X 110, Y 88, Z 12} c_vel
LIN {X 110, Y 81, Z 12} c_vel
LIN {X 111, Y 74, Z 12} c_vel
LIN {X 113, Y 69, Z 12} c_vel
LIN {X 116, Y 63, Z 12} c_vel
LIN {X 119, Y 58, Z 12} c_vel
LIN {X 124, Y 53, Z 12} c_vel
LIN {X 130, Y 48, Z 12} c_vel
LIN {X 138, Y 43, Z 12} c_vel
LIN {X 111, Y 0, Z 12} c_vel
$OUT[4] = FALSE
WAIT SEC 10.0
LIN {X 111, Y 0, Z 13} c_vel
$OUT[4] = TRUE
LIN {X 111, Y 0, Z 13} c_vel
LIN {X 106, Y 3, Z 13} c_vel
LIN {X 97, Y 9, Z 13} c_vel
LIN {X 89, Y 16, Z 13} c_vel
LIN {X 83, Y 23, Z 13} c_vel
LIN {X 77, Y 31, Z 13} c_vel
LIN {X 71, Y 39, Z 13} c_vel
LIN {X 67, Y 47, Z 13} c_vel
LIN {X 64, Y 56, Z 13} c_vel
LIN {X 62, Y 64, Z 13} c_vel
LIN {X 60, Y 73, Z 13} c_vel
LIN {X 59, Y 82, Z 13} c_vel
LIN {X 59, Y 92, Z 13} c_vel
LIN {X 60, Y 103, Z 13} c_vel
LIN {X 62, Y 114, Z 13} c_vel
LIN {X 65, Y 127, Z 13} c_vel
LIN {X 69, Y 144, Z 13} c_vel
LIN {X 74, Y 163, Z 13} c_vel
LIN {X 79, Y 180, Z 13} c_vel
LIN {X 81, Y 191, Z 13} c_vel
LIN {X 82, Y 201, Z 13} c_vel
LIN {X 82, Y 209, Z 13} c_vel
LIN {X 82, Y 217, Z 13} c_vel
LIN {X 80, Y 223, Z 13} c_vel
LIN {X 78, Y 229, Z 13} c_vel
LIN {X 75, Y 234, Z 13} c_vel
LIN {X 71, Y 240, Z 13} c_vel
LIN {X 66, Y 245, Z 13} c_vel
LIN {X 60, Y 250, Z 13} c_vel
LIN {X 52, Y 256, Z 13} c_vel
LIN {X 42, Y 261, Z 13} c_vel
LIN {X 30, Y 267, Z 13} c_vel
LIN {X 16, Y 273, Z 13} c_vel
LIN {X 0, Y 278, Z 13} c_vel
LIN {X 14, Y 327, Z 13} c_vel
LIN {X 28, Y 322, Z 13} c_vel
LIN {X 43, Y 317, Z 13} c_vel
LIN {X 57, Y 311, Z 13} c_vel
LIN {X 70, Y 304, Z 13} c_vel
LIN {X 81, Y 298, Z 13} c_vel
LIN {X 90, Y 291, Z 13} c_vel
LIN {X 99, Y 284, Z 13} c_vel
LIN {X 106, Y 277, Z 13} c_vel
LIN {X 113, Y 269, Z 13} c_vel
LIN {X 118, Y 261, Z 13} c_vel
LIN {X 123, Y 253, Z 13} c_vel
LIN {X 127, Y 244, Z 13} c_vel
LIN {X 130, Y 235, Z 13} c_vel
LIN {X 131, Y 226, Z 13} c_vel
LIN {X 133, Y 217, Z 13} c_vel
LIN {X 133, Y 207, Z 13} c_vel
LIN {X 133, Y 197, Z 13} c_vel
LIN {X 131, Y 186, Z 13} c_vel
LIN {X 129, Y 173, Z 13} c_vel
LIN {X 126, Y 160, Z 13} c_vel
LIN {X 120, Y 138, Z 13} c_vel
LIN {X 115, Y 118, Z 13} c_vel
LIN {X 112, Y 106, Z 13} c_vel
LIN {X 111, Y 96, Z 13} c_vel
LIN {X 110, Y 88, Z 13} c_vel
LIN {X 110, Y 81, Z 13} c_vel
LIN {X 111, Y 74, Z 13} c_vel
LIN {X 113, Y 69, Z 13} c_vel
LIN {X 116, Y 63, Z 13} c_vel
LIN {X 119, Y 58, Z 13} c_vel
LIN {X 124, Y 53, Z 13} c_vel
LIN {X 130, Y 48, Z 13} c_vel
LIN {X 138, Y 43, Z 13} c_vel
LIN {X 111, Y 0, Z 13} c_vel
$OUT[4] = FALSE
WAIT SEC 10.0
LIN {X 111, Y 0, Z 14} c_vel
$OUT[4] = TRUE
LIN {X 111, Y 0, Z 14} c_vel
LIN {X 106, Y 3, Z 14} c_vel
LIN {X 97, Y 9, Z 14} c_vel
LIN {X 89, Y 16, Z 14} c_vel
LIN {X 83, Y 23, Z 14} c_vel
LIN {X 77, Y 31, Z 14} c_vel
LIN {X 71, Y 39, Z 14} c_vel
LIN {X 67, Y 47, Z 14} c_vel
LIN {X 64, Y 56, Z 14} c_vel
LIN {X 62, Y 64, Z 14} c_vel
LIN {X 60, Y 73, Z 14} c_vel
LIN {X 59, Y 82, Z 14} c_vel
LIN {X 59, Y 92, Z 14} c_vel
LIN {X 60, Y 103, Z 14} c_vel
LIN {X 62, Y 114, Z 14} c_vel
LIN {X 65, Y 127, Z 14} c_vel
LIN {X 69, Y 144, Z 14} c_vel
LIN {X 74, Y 163, Z 14} c_vel
LIN {X 79, Y 180, Z 14} c_vel
LIN {X 81, Y 191, Z 14} c_vel
LIN {X 82, Y 201, Z 14} c_vel
LIN {X 82, Y 209, Z 14} c_vel
LIN {X 82, Y 217, Z 14} c_vel
LIN {X 80, Y 223, Z 14} c_vel
LIN {X 78, Y 229, Z 14} c_vel
LIN {X 75, Y 234, Z 14} c_vel
LIN {X 71, Y 240, Z 14} c_vel
LIN {X 66, Y 245, Z 14} c_vel
LIN {X 60, Y 250, Z 14} c_vel
LIN {X 52, Y 256, Z 14} c_vel
LIN {X 42, Y 261, Z 14} c_vel
LIN {X 30, Y 267, Z 14} c_vel
LIN {X 16, Y 273, Z 14} c_vel
LIN {X 0, Y 278, Z 14} c_vel
LIN {X 14, Y 327, Z 14} c_vel
LIN {X 28, Y 322, Z 14} c_vel
LIN {X 43, Y 317, Z 14} c_vel
LIN {X 57, Y 311, Z 14} c_vel
LIN {X 70, Y 304, Z 14} c_vel
LIN {X 81, Y 298, Z 14} c_vel
LIN {X 90, Y 291, Z 14} c_vel
LIN {X 99, Y 284, Z 14} c_vel
LIN {X 106, Y 277, Z 14} c_vel
LIN {X 113, Y 269, Z 14} c_vel
LIN {X 118, Y 261, Z 14} c_vel
LIN {X 123, Y 253, Z 14} c_vel
LIN {X 127, Y 244, Z 14} c_vel
LIN {X 130, Y 235, Z 14} c_vel
LIN {X 131, Y 226, Z 14} c_vel
LIN {X 133, Y 217, Z 14} c_vel
LIN {X 133, Y 207, Z 14} c_vel
LIN {X 133, Y 197, Z 14} c_vel
LIN {X 131, Y 186, Z 14} c_vel
LIN {X 129, Y 173, Z 14} c_vel
LIN {X 126, Y 160, Z 14} c_vel
LIN {X 120, Y 138, Z 14} c_vel
LIN {X 115, Y 118, Z 14} c_vel
LIN {X 112, Y 106, Z 14} c_vel
LIN {X 111, Y 96, Z 14} c_vel
LIN {X 110, Y 88, Z 14} c_vel
LIN {X 110, Y 81, Z 14} c_vel
LIN {X 111, Y 74, Z 14} c_vel
LIN {X 113, Y 69, Z 14} c_vel
LIN {X 116, Y 63, Z 14} c_vel
LIN {X 119, Y 58, Z 14} c_vel
LIN {X 124, Y 53, Z 14} c_vel
LIN {X 130, Y 48, Z 14} c_vel
LIN {X 138, Y 43, Z 14} c_vel
LIN {X 111, Y 0, Z 14} c_vel
$OUT[4] = FALSE
WAIT SEC 10.0
LIN {X 111, Y 0, Z 15} c_vel
$OUT[4] = TRUE
LIN {X 111, Y 0, Z 15} c_vel
LIN {X 106, Y 3, Z 15} c_vel
LIN {X 97, Y 9, Z 15} c_vel
LIN {X 89, Y 16, Z 15} c_vel
LIN {X 83, Y 23, Z 15} c_vel
LIN {X 77, Y 31, Z 15} c_vel
LIN {X 71, Y 39, Z 15} c_vel
LIN {X 67, Y 47, Z 15} c_vel
LIN {X 64, Y 56, Z 15} c_vel
LIN {X 62, Y 64, Z 15} c_vel
LIN {X 60, Y 73, Z 15} c_vel
LIN {X 59, Y 82, Z 15} c_vel
LIN {X 59, Y 92, Z 15} c_vel
LIN {X 60, Y 103, Z 15} c_vel
LIN {X 62, Y 114, Z 15} c_vel
LIN {X 65, Y 127, Z 15} c_vel
LIN {X 69, Y 144, Z 15} c_vel
LIN {X 74, Y 163, Z 15} c_vel
LIN {X 79, Y 180, Z 15} c_vel
LIN {X 81, Y 191, Z 15} c_vel
LIN {X 82, Y 201, Z 15} c_vel
LIN {X 82, Y 209, Z 15} c_vel
LIN {X 82, Y 217, Z 15} c_vel
LIN {X 80, Y 223, Z 15} c_vel
LIN {X 78, Y 229, Z 15} c_vel
LIN {X 75, Y 234, Z 15} c_vel
LIN {X 71, Y 240, Z 15} c_vel
LIN {X 66, Y 245, Z 15} c_vel
LIN {X 60, Y 250, Z 15} c_vel
LIN {X 52, Y 256, Z 15} c_vel
LIN {X 42, Y 261, Z 15} c_vel
LIN {X 30, Y 267, Z 15} c_vel
LIN {X 16, Y 273, Z 15} c_vel
LIN {X 0, Y 278, Z 15} c_vel
LIN {X 14, Y 327, Z 15} c_vel
LIN {X 28, Y 322, Z 15} c_vel
LIN {X 43, Y 317, Z 15} c_vel
LIN {X 57, Y 311, Z 15} c_vel
LIN {X 70, Y 304, Z 15} c_vel
LIN {X 81, Y 298, Z 15} c_vel
LIN {X 90, Y 291, Z 15} c_vel
LIN {X 99, Y 284, Z 15} c_vel
LIN {X 106, Y 277, Z 15} c_vel
LIN {X 113, Y 269, Z 15} c_vel
LIN {X 118, Y 261, Z 15} c_vel
LIN {X 123, Y 253, Z 15} c_vel
LIN {X 127, Y 244, Z 15} c_vel
LIN {X 130, Y 235, Z 15} c_vel
LIN {X 131, Y 226, Z 15} c_vel
LIN {X 133, Y 217, Z 15} c_vel
LIN {X 133, Y 207, Z 15} c_vel
LIN {X 133, Y 197, Z 15} c_vel
LIN {X 131, Y 186, Z 15} c_vel
LIN {X 129, Y 173, Z 15} c_vel
LIN {X 126, Y 160, Z 15} c_vel
LIN {X 120, Y 138, Z 15} c_vel
LIN {X 115, Y 118, Z 15} c_vel
LIN {X 112, Y 106, Z 15} c_vel
LIN {X 111, Y 96, Z 15} c_vel
LIN {X 110, Y 88, Z 15} c_vel
LIN {X 110, Y 81, Z 15} c_vel
LIN {X 111, Y 74, Z 15} c_vel
LIN {X 113, Y 69, Z 15} c_vel
LIN {X 116, Y 63, Z 15} c_vel
LIN {X 119, Y 58, Z 15} c_vel
LIN {X 124, Y 53, Z 15} c_vel
LIN {X 130, Y 48, Z 15} c_vel
LIN {X 138, Y 43, Z 15} c_vel
LIN {X 111, Y 0, Z 15} c_vel
$OUT[4] = FALSE
WAIT SEC 10.0
LIN {X 111, Y 0, Z 16} c_vel
$OUT[4] = TRUE
LIN {X 111, Y 0, Z 16} c_vel
LIN {X 106, Y 3, Z 16} c_vel
LIN {X 97, Y 9, Z 16} c_vel
LIN {X 89, Y 16, Z 16} c_vel
LIN {X 83, Y 23, Z 16} c_vel
LIN {X 77, Y 31, Z 16} c_vel
LIN {X 71, Y 39, Z 16} c_vel
LIN {X 67, Y 47, Z 16} c_vel
LIN {X 64, Y 56, Z 16} c_vel
LIN {X 62, Y 64, Z 16} c_vel
LIN {X 60, Y 73, Z 16} c_vel
LIN {X 59, Y 82, Z 16} c_vel
LIN {X 59, Y 92, Z 16} c_vel
LIN {X 60, Y 103, Z 16} c_vel
LIN {X 62, Y 114, Z 16} c_vel
LIN {X 65, Y 127, Z 16} c_vel
LIN {X 69, Y 144, Z 16} c_vel
LIN {X 74, Y 163, Z 16} c_vel
LIN {X 79, Y 180, Z 16} c_vel
LIN {X 81, Y 191, Z 16} c_vel
LIN {X 82, Y 201, Z 16} c_vel
LIN {X 82, Y 209, Z 16} c_vel
LIN {X 82, Y 217, Z 16} c_vel
LIN {X 80, Y 223, Z 16} c_vel
LIN {X 78, Y 229, Z 16} c_vel
LIN {X 75, Y 234, Z 16} c_vel
LIN {X 71, Y 240, Z 16} c_vel
LIN {X 66, Y 245, Z 16} c_vel
LIN {X 60, Y 250, Z 16} c_vel
LIN {X 52, Y 256, Z 16} c_vel
LIN {X 42, Y 261, Z 16} c_vel
LIN {X 30, Y 267, Z 16} c_vel
LIN {X 16, Y 273, Z 16} c_vel
LIN {X 0, Y 278, Z 16} c_vel
LIN {X 14, Y 327, Z 16} c_vel
LIN {X 28, Y 322, Z 16} c_vel
LIN {X 43, Y 317, Z 16} c_vel
LIN {X 57, Y 311, Z 16} c_vel
LIN {X 70, Y 304, Z 16} c_vel
LIN {X 81, Y 298, Z 16} c_vel
LIN {X 90, Y 291, Z 16} c_vel
LIN {X 99, Y 284, Z 16} c_vel
LIN {X 106, Y 277, Z 16} c_vel
LIN {X 113, Y 269, Z 16} c_vel
LIN {X 118, Y 261, Z 16} c_vel
LIN {X 123, Y 253, Z 16} c_vel
LIN {X 127, Y 244, Z 16} c_vel
LIN {X 130, Y 235, Z 16} c_vel
LIN {X 131, Y 226, Z 16} c_vel
LIN {X 133, Y 217, Z 16} c_vel
LIN {X 133, Y 207, Z 16} c_vel
LIN {X 133, Y 197, Z 16} c_vel
LIN {X 131, Y 186, Z 16} c_vel
LIN {X 129, Y 173, Z 16} c_vel
LIN {X 126, Y 160, Z 16} c_vel
LIN {X 120, Y 138, Z 16} c_vel
LIN {X 115, Y 118, Z 16} c_vel
LIN {X 112, Y 106, Z 16} c_vel
LIN {X 111, Y 96, Z 16} c_vel
LIN {X 110, Y 88, Z 16} c_vel
LIN {X 110, Y 81, Z 16} c_vel
LIN {X 111, Y 74, Z 16} c_vel
LIN {X 113, Y 69, Z 16} c_vel
LIN {X 116, Y 63, Z 16} c_vel
LIN {X 119, Y 58, Z 16} c_vel
LIN {X 124, Y 53, Z 16} c_vel
LIN {X 130, Y 48, Z 16} c_vel
LIN {X 138, Y 43, Z 16} c_vel
LIN {X 111, Y 0, Z 16} c_vel
$OUT[4] = FALSE
WAIT SEC 10.0
LIN {X 111, Y 0, Z 17} c_vel
$OUT[4] = TRUE
LIN {X 111, Y 0, Z 17} c_vel
LIN {X 106, Y 3, Z 17} c_vel
LIN {X 97, Y 9, Z 17} c_vel
LIN {X 89, Y 16, Z 17} c_vel
LIN {X 83, Y 23, Z 17} c_vel
LIN {X 77, Y 31, Z 17} c_vel
LIN {X 71, Y 39, Z 17} c_vel
LIN {X 67, Y 47, Z 17} c_vel
LIN {X 64, Y 56, Z 17} c_vel
LIN {X 62, Y 64, Z 17} c_vel
LIN {X 60, Y 73, Z 17} c_vel
LIN {X 59, Y 82, Z 17} c_vel
LIN {X 59, Y 92, Z 17} c_vel
LIN {X 60, Y 103, Z 17} c_vel
LIN {X 62, Y 114, Z 17} c_vel
LIN {X 65, Y 127, Z 17} c_vel
LIN {X 69, Y 144, Z 17} c_vel
LIN {X 74, Y 163, Z 17} c_vel
LIN {X 79, Y 180, Z 17} c_vel
LIN {X 81, Y 191, Z 17} c_vel
LIN {X 82, Y 201, Z 17} c_vel
LIN {X 82, Y 209, Z 17} c_vel
LIN {X 82, Y 217, Z 17} c_vel
LIN {X 80, Y 223, Z 17} c_vel
LIN {X 78, Y 229, Z 17} c_vel
LIN {X 75, Y 234, Z 17} c_vel
LIN {X 71, Y 240, Z 17} c_vel
LIN {X 66, Y 245, Z 17} c_vel
LIN {X 60, Y 250, Z 17} c_vel
LIN {X 52, Y 256, Z 17} c_vel
LIN {X 42, Y 261, Z 17} c_vel
LIN {X 30, Y 267, Z 17} c_vel
LIN {X 16, Y 273, Z 17} c_vel
LIN {X 0, Y 278, Z 17} c_vel
LIN {X 14, Y 327, Z 17} c_vel
LIN {X 28, Y 322, Z 17} c_vel
LIN {X 43, Y 317, Z 17} c_vel
LIN {X 57, Y 311, Z 17} c_vel
LIN {X 70, Y 304, Z 17} c_vel
LIN {X 81, Y 298, Z 17} c_vel
LIN {X 90, Y 291, Z 17} c_vel
LIN {X 99, Y 284, Z 17} c_vel
LIN {X 106, Y 277, Z 17} c_vel
LIN {X 113, Y 269, Z 17} c_vel
LIN {X 118, Y 261, Z 17} c_vel
LIN {X 123, Y 253, Z 17} c_vel
LIN {X 127, Y 244, Z 17} c_vel
LIN {X 130, Y 235, Z 17} c_vel
LIN {X 131, Y 226, Z 17} c_vel
LIN {X 133, Y 217, Z 17} c_vel
LIN {X 133, Y 207, Z 17} c_vel
LIN {X 133, Y 197, Z 17} c_vel
LIN {X 131, Y 186, Z 17} c_vel
LIN {X 129, Y 173, Z 17} c_vel
LIN {X 126, Y 160, Z 17} c_vel
LIN {X 120, Y 138, Z 17} c_vel
LIN {X 115, Y 118, Z 17} c_vel
LIN {X 112, Y 106, Z 17} c_vel
LIN {X 111, Y 96, Z 17} c_vel
LIN {X 110, Y 88, Z 17} c_vel
LIN {X 110, Y 81, Z 17} c_vel
LIN {X 111, Y 74, Z 17} c_vel
LIN {X 113, Y 69, Z 17} c_vel
LIN {X 116, Y 63, Z 17} c_vel
LIN {X 119, Y 58, Z 17} c_vel
LIN {X 124, Y 53, Z 17} c_vel
LIN {X 130, Y 48, Z 17} c_vel
LIN {X 138, Y 43, Z 17} c_vel
LIN {X 111, Y 0, Z 17} c_vel
$OUT[4] = FALSE
WAIT SEC 10.0
LIN {X 111, Y 0, Z 18} c_vel
$OUT[4] = TRUE
LIN {X 111, Y 0, Z 18} c_vel
LIN {X 106, Y 3, Z 18} c_vel
LIN {X 97, Y 9, Z 18} c_vel
LIN {X 89, Y 16, Z 18} c_vel
LIN {X 83, Y 23, Z 18} c_vel
LIN {X 77, Y 31, Z 18} c_vel
LIN {X 71, Y 39, Z 18} c_vel
LIN {X 67, Y 47, Z 18} c_vel
LIN {X 64, Y 56, Z 18} c_vel
LIN {X 62, Y 64, Z 18} c_vel
LIN {X 60, Y 73, Z 18} c_vel
LIN {X 59, Y 82, Z 18} c_vel
LIN {X 59, Y 92, Z 18} c_vel
LIN {X 60, Y 103, Z 18} c_vel
LIN {X 62, Y 114, Z 18} c_vel
LIN {X 65, Y 127, Z 18} c_vel
LIN {X 69, Y 144, Z 18} c_vel
LIN {X 74, Y 163, Z 18} c_vel
LIN {X 79, Y 180, Z 18} c_vel
LIN {X 81, Y 191, Z 18} c_vel
LIN {X 82, Y 201, Z 18} c_vel
LIN {X 82, Y 209, Z 18} c_vel
LIN {X 82, Y 217, Z 18} c_vel
LIN {X 80, Y 223, Z 18} c_vel
LIN {X 78, Y 229, Z 18} c_vel
LIN {X 75, Y 234, Z 18} c_vel
LIN {X 71, Y 240, Z 18} c_vel
LIN {X 66, Y 245, Z 18} c_vel
LIN {X 60, Y 250, Z 18} c_vel
LIN {X 52, Y 256, Z 18} c_vel
LIN {X 42, Y 261, Z 18} c_vel
LIN {X 30, Y 267, Z 18} c_vel
LIN {X 16, Y 273, Z 18} c_vel
LIN {X 0, Y 278, Z 18} c_vel
LIN {X 14, Y 327, Z 18} c_vel
LIN {X 28, Y 322, Z 18} c_vel
LIN {X 43, Y 317, Z 18} c_vel
LIN {X 57, Y 311, Z 18} c_vel
LIN {X 70, Y 304, Z 18} c_vel
LIN {X 81, Y 298, Z 18} c_vel
LIN {X 90, Y 291, Z 18} c_vel
LIN {X 99, Y 284, Z 18} c_vel
LIN {X 106, Y 277, Z 18} c_vel
LIN {X 113, Y 269, Z 18} c_vel
LIN {X 118, Y 261, Z 18} c_vel
LIN {X 123, Y 253, Z 18} c_vel
LIN {X 127, Y 244, Z 18} c_vel
LIN {X 130, Y 235, Z 18} c_vel
LIN {X 131, Y 226, Z 18} c_vel
LIN {X 133, Y 217, Z 18} c_vel
LIN {X 133, Y 207, Z 18} c_vel
LIN {X 133, Y 197, Z 18} c_vel
LIN {X 131, Y 186, Z 18} c_vel
LIN {X 129, Y 173, Z 18} c_vel
LIN {X 126, Y 160, Z 18} c_vel
LIN {X 120, Y 138, Z 18} c_vel
LIN {X 115, Y 118, Z 18} c_vel
LIN {X 112, Y 106, Z 18} c_vel
LIN {X 111, Y 96, Z 18} c_vel
LIN {X 110, Y 88, Z 18} c_vel
LIN {X 110, Y 81, Z 18} c_vel
LIN {X 111, Y 74, Z 18} c_vel
LIN {X 113, Y 69, Z 18} c_vel
LIN {X 116, Y 63, Z 18} c_vel
LIN {X 119, Y 58, Z 18} c_vel
LIN {X 124, Y 53, Z 18} c_vel
LIN {X 130, Y 48, Z 18} c_vel
LIN {X 138, Y 43, Z 18} c_vel
LIN {X 111, Y 0, Z 18} c_vel
$OUT[4] = FALSE
WAIT SEC 10.0
LIN {X 111, Y 0, Z 19} c_vel
$OUT[4] = TRUE
LIN {X 111, Y 0, Z 19} c_vel
LIN {X 106, Y 3, Z 19} c_vel
LIN {X 97, Y 9, Z 19} c_vel
LIN {X 89, Y 16, Z 19} c_vel
LIN {X 83, Y 23, Z 19} c_vel
LIN {X 77, Y 31, Z 19} c_vel
LIN {X 71, Y 39, Z 19} c_vel
LIN {X 67, Y 47, Z 19} c_vel
LIN {X 64, Y 56, Z 19} c_vel
LIN {X 62, Y 64, Z 19} c_vel
LIN {X 60, Y 73, Z 19} c_vel
LIN {X 59, Y 82, Z 19} c_vel
LIN {X 59, Y 92, Z 19} c_vel
LIN {X 60, Y 103, Z 19} c_vel
LIN {X 62, Y 114, Z 19} c_vel
LIN {X 65, Y 127, Z 19} c_vel
LIN {X 69, Y 144, Z 19} c_vel
LIN {X 74, Y 163, Z 19} c_vel
LIN {X 79, Y 180, Z 19} c_vel
LIN {X 81, Y 191, Z 19} c_vel
LIN {X 82, Y 201, Z 19} c_vel
LIN {X 82, Y 209, Z 19} c_vel
LIN {X 82, Y 217, Z 19} c_vel
LIN {X 80, Y 223, Z 19} c_vel
LIN {X 78, Y 229, Z 19} c_vel
LIN {X 75, Y 234, Z 19} c_vel
LIN {X 71, Y 240, Z 19} c_vel
LIN {X 66, Y 245, Z 19} c_vel
LIN {X 60, Y 250, Z 19} c_vel
LIN {X 52, Y 256, Z 19} c_vel
LIN {X 42, Y 261, Z 19} c_vel
LIN {X 30, Y 267, Z 19} c_vel
LIN {X 16, Y 273, Z 19} c_vel
LIN {X 0, Y 278, Z 19} c_vel
LIN {X 14, Y 327, Z 19} c_vel
LIN {X 28, Y 322, Z 19} c_vel
LIN {X 43, Y 317, Z 19} c_vel
LIN {X 57, Y 311, Z 19} c_vel
LIN {X 70, Y 304, Z 19} c_vel
LIN {X 81, Y 298, Z 19} c_vel
LIN {X 90, Y 291, Z 19} c_vel
LIN {X 99, Y 284, Z 19} c_vel
LIN {X 106, Y 277, Z 19} c_vel
LIN {X 113, Y 269, Z 19} c_vel
LIN {X 118, Y 261, Z 19} c_vel
LIN {X 123, Y 253, Z 19} c_vel
LIN {X 127, Y 244, Z 19} c_vel
LIN {X 130, Y 235, Z 19} c_vel
LIN {X 131, Y 226, Z 19} c_vel
LIN {X 133, Y 217, Z 19} c_vel
LIN {X 133, Y 207, Z 19} c_vel
LIN {X 133, Y 197, Z 19} c_vel
LIN {X 131, Y 186, Z 19} c_vel
LIN {X 129, Y 173, Z 19} c_vel
LIN {X 126, Y 160, Z 19} c_vel
LIN {X 120, Y 138, Z 19} c_vel
LIN {X 115, Y 118, Z 19} c_vel
LIN {X 112, Y 106, Z 19} c_vel
LIN {X 111, Y 96, Z 19} c_vel
LIN {X 110, Y 88, Z 19} c_vel
LIN {X 110, Y 81, Z 19} c_vel
LIN {X 111, Y 74, Z 19} c_vel
LIN {X 113, Y 69, Z 19} c_vel
LIN {X 116, Y 63, Z 19} c_vel
LIN {X 119, Y 58, Z 19} c_vel
LIN {X 124, Y 53, Z 19} c_vel
LIN {X 130, Y 48, Z 19} c_vel
LIN {X 138, Y 43, Z 19} c_vel
LIN {X 111, Y 0, Z 19} c_vel
$OUT[4] = FALSE
WAIT SEC 10.0
LIN {X 111, Y 0, Z 20} c_vel
$OUT[4] = TRUE
LIN {X 111, Y 0, Z 20} c_vel
LIN {X 106, Y 3, Z 20} c_vel
LIN {X 97, Y 9, Z 20} c_vel
LIN {X 89, Y 16, Z 20} c_vel
LIN {X 83, Y 23, Z 20} c_vel
LIN {X 77, Y 31, Z 20} c_vel
LIN {X 71, Y 39, Z 20} c_vel
LIN {X 67, Y 47, Z 20} c_vel
LIN {X 64, Y 56, Z 20} c_vel
LIN {X 62, Y 64, Z 20} c_vel
LIN {X 60, Y 73, Z 20} c_vel
LIN {X 59, Y 82, Z 20} c_vel
LIN {X 59, Y 92, Z 20} c_vel
LIN {X 60, Y 103, Z 20} c_vel
LIN {X 62, Y 114, Z 20} c_vel
LIN {X 65, Y 127, Z 20} c_vel
LIN {X 69, Y 144, Z 20} c_vel
LIN {X 74, Y 163, Z 20} c_vel
LIN {X 79, Y 180, Z 20} c_vel
LIN {X 81, Y 191, Z 20} c_vel
LIN {X 82, Y 201, Z 20} c_vel
LIN {X 82, Y 209, Z 20} c_vel
LIN {X 82, Y 217, Z 20} c_vel
LIN {X 80, Y 223, Z 20} c_vel
LIN {X 78, Y 229, Z 20} c_vel
LIN {X 75, Y 234, Z 20} c_vel
LIN {X 71, Y 240, Z 20} c_vel
LIN {X 66, Y 245, Z 20} c_vel
LIN {X 60, Y 250, Z 20} c_vel
LIN {X 52, Y 256, Z 20} c_vel
LIN {X 42, Y 261, Z 20} c_vel
LIN {X 30, Y 267, Z 20} c_vel
LIN {X 16, Y 273, Z 20} c_vel
LIN {X 0, Y 278, Z 20} c_vel
LIN {X 14, Y 327, Z 20} c_vel
LIN {X 28, Y 322, Z 20} c_vel
LIN {X 43, Y 317, Z 20} c_vel
LIN {X 57, Y 311, Z 20} c_vel
LIN {X 70, Y 304, Z 20} c_vel
LIN {X 81, Y 298, Z 20} c_vel
LIN {X 90, Y 291, Z 20} c_vel
LIN {X 99, Y 284, Z 20} c_vel
LIN {X 106, Y 277, Z 20} c_vel
LIN {X 113, Y 269, Z 20} c_vel
LIN {X 118, Y 261, Z 20} c_vel
LIN {X 123, Y 253, Z 20} c_vel
LIN {X 127, Y 244, Z 20} c_vel
LIN {X 130, Y 235, Z 20} c_vel
LIN {X 131, Y 226, Z 20} c_vel
LIN {X 133, Y 217, Z 20} c_vel
LIN {X 133, Y 207, Z 20} c_vel
LIN {X 133, Y 197, Z 20} c_vel
LIN {X 131, Y 186, Z 20} c_vel
LIN {X 129, Y 173, Z 20} c_vel
LIN {X 126, Y 160, Z 20} c_vel
LIN {X 120, Y 138, Z 20} c_vel
LIN {X 115, Y 118, Z 20} c_vel
LIN {X 112, Y 106, Z 20} c_vel
LIN {X 111, Y 96, Z 20} c_vel
LIN {X 110, Y 88, Z 20} c_vel
LIN {X 110, Y 81, Z 20} c_vel
LIN {X 111, Y 74, Z 20} c_vel
LIN {X 113, Y 69, Z 20} c_vel
LIN {X 116, Y 63, Z 20} c_vel
LIN {X 119, Y 58, Z 20} c_vel
LIN {X 124, Y 53, Z 20} c_vel
LIN {X 130, Y 48, Z 20} c_vel
LIN {X 138, Y 43, Z 20} c_vel
LIN {X 111, Y 0, Z 20} c_vel
$OUT[4] = FALSE
WAIT SEC 10.0
LIN {X 111, Y 0, Z 21} c_vel
$OUT[4] = TRUE
LIN {X 111, Y 0, Z 21} c_vel
LIN {X 106, Y 3, Z 21} c_vel
LIN {X 97, Y 9, Z 21} c_vel
LIN {X 89, Y 16, Z 21} c_vel
LIN {X 83, Y 23, Z 21} c_vel
LIN {X 77, Y 31, Z 21} c_vel
LIN {X 71, Y 39, Z 21} c_vel
LIN {X 67, Y 47, Z 21} c_vel
LIN {X 64, Y 56, Z 21} c_vel
LIN {X 62, Y 64, Z 21} c_vel
LIN {X 60, Y 73, Z 21} c_vel
LIN {X 59, Y 82, Z 21} c_vel
LIN {X 59, Y 92, Z 21} c_vel
LIN {X 60, Y 103, Z 21} c_vel
LIN {X 62, Y 114, Z 21} c_vel
LIN {X 65, Y 127, Z 21} c_vel
LIN {X 69, Y 144, Z 21} c_vel
LIN {X 74, Y 163, Z 21} c_vel
LIN {X 79, Y 180, Z 21} c_vel
LIN {X 81, Y 191, Z 21} c_vel
LIN {X 82, Y 201, Z 21} c_vel
LIN {X 82, Y 209, Z 21} c_vel
LIN {X 82, Y 217, Z 21} c_vel
LIN {X 80, Y 223, Z 21} c_vel
LIN {X 78, Y 229, Z 21} c_vel
LIN {X 75, Y 234, Z 21} c_vel
LIN {X 71, Y 240, Z 21} c_vel
LIN {X 66, Y 245, Z 21} c_vel
LIN {X 60, Y 250, Z 21} c_vel
LIN {X 52, Y 256, Z 21} c_vel
LIN {X 42, Y 261, Z 21} c_vel
LIN {X 30, Y 267, Z 21} c_vel
LIN {X 16, Y 273, Z 21} c_vel
LIN {X 0, Y 278, Z 21} c_vel
LIN {X 14, Y 327, Z 21} c_vel
LIN {X 28, Y 322, Z 21} c_vel
LIN {X 43, Y 317, Z 21} c_vel
LIN {X 57, Y 311, Z 21} c_vel
LIN {X 70, Y 304, Z 21} c_vel
LIN {X 81, Y 298, Z 21} c_vel
LIN {X 90, Y 291, Z 21} c_vel
LIN {X 99, Y 284, Z 21} c_vel
LIN {X 106, Y 277, Z 21} c_vel
LIN {X 113, Y 269, Z 21} c_vel
LIN {X 118, Y 261, Z 21} c_vel
LIN {X 123, Y 253, Z 21} c_vel
LIN {X 127, Y 244, Z 21} c_vel
LIN {X 130, Y 235, Z 21} c_vel
LIN {X 131, Y 226, Z 21} c_vel
LIN {X 133, Y 217, Z 21} c_vel
LIN {X 133, Y 207, Z 21} c_vel
LIN {X 133, Y 197, Z 21} c_vel
LIN {X 131, Y 186, Z 21} c_vel
LIN {X 129, Y 173, Z 21} c_vel
LIN {X 126, Y 160, Z 21} c_vel
LIN {X 120, Y 138, Z 21} c_vel
LIN {X 115, Y 118, Z 21} c_vel
LIN {X 112, Y 106, Z 21} c_vel
LIN {X 111, Y 96, Z 21} c_vel
LIN {X 110, Y 88, Z 21} c_vel
LIN {X 110, Y 81, Z 21} c_vel
LIN {X 111, Y 74, Z 21} c_vel
LIN {X 113, Y 69, Z 21} c_vel
LIN {X 116, Y 63, Z 21} c_vel
LIN {X 119, Y 58, Z 21} c_vel
LIN {X 124, Y 53, Z 21} c_vel
LIN {X 130, Y 48, Z 21} c_vel
LIN {X 138, Y 43, Z 21} c_vel
LIN {X 111, Y 0, Z 21} c_vel
$OUT[4] = FALSE
WAIT SEC 10.0
LIN {X 111, Y 0, Z 22} c_vel
$OUT[4] = TRUE
LIN {X 111, Y 0, Z 22} c_vel
LIN {X 106, Y 3, Z 22} c_vel
LIN {X 97, Y 9, Z 22} c_vel
LIN {X 89, Y 16, Z 22} c_vel
LIN {X 83, Y 23, Z 22} c_vel
LIN {X 77, Y 31, Z 22} c_vel
LIN {X 71, Y 39, Z 22} c_vel
LIN {X 67, Y 47, Z 22} c_vel
LIN {X 64, Y 56, Z 22} c_vel
LIN {X 62, Y 64, Z 22} c_vel
LIN {X 60, Y 73, Z 22} c_vel
LIN {X 59, Y 82, Z 22} c_vel
LIN {X 59, Y 92, Z 22} c_vel
LIN {X 60, Y 103, Z 22} c_vel
LIN {X 62, Y 114, Z 22} c_vel
LIN {X 65, Y 127, Z 22} c_vel
LIN {X 69, Y 144, Z 22} c_vel
LIN {X 74, Y 163, Z 22} c_vel
LIN {X 79, Y 180, Z 22} c_vel
LIN {X 81, Y 191, Z 22} c_vel
LIN {X 82, Y 201, Z 22} c_vel
LIN {X 82, Y 209, Z 22} c_vel
LIN {X 82, Y 217, Z 22} c_vel
LIN {X 80, Y 223, Z 22} c_vel
LIN {X 78, Y 229, Z 22} c_vel
LIN {X 75, Y 234, Z 22} c_vel
LIN {X 71, Y 240, Z 22} c_vel
LIN {X 66, Y 245, Z 22} c_vel
LIN {X 60, Y 250, Z 22} c_vel
LIN {X 52, Y 256, Z 22} c_vel
LIN {X 42, Y 261, Z 22} c_vel
LIN {X 30, Y 267, Z 22} c_vel
LIN {X 16, Y 273, Z 22} c_vel
LIN {X 0, Y 278, Z 22} c_vel
LIN {X 14, Y 327, Z 22} c_vel
LIN {X 28, Y 322, Z 22} c_vel
LIN {X 43, Y 317, Z 22} c_vel
LIN {X 57, Y 311, Z 22} c_vel
LIN {X 70, Y 304, Z 22} c_vel
LIN {X 81, Y 298, Z 22} c_vel
LIN {X 90, Y 291, Z 22} c_vel
LIN {X 99, Y 284, Z 22} c_vel
LIN {X 106, Y 277, Z 22} c_vel
LIN {X 113, Y 269, Z 22} c_vel
LIN {X 118, Y 261, Z 22} c_vel
LIN {X 123, Y 253, Z 22} c_vel
LIN {X 127, Y 244, Z 22} c_vel
LIN {X 130, Y 235, Z 22} c_vel
LIN {X 131, Y 226, Z 22} c_vel
LIN {X 133, Y 217, Z 22} c_vel
LIN {X 133, Y 207, Z 22} c_vel
LIN {X 133, Y 197, Z 22} c_vel
LIN {X 131, Y 186, Z 22} c_vel
LIN {X 129, Y 173, Z 22} c_vel
LIN {X 126, Y 160, Z 22} c_vel
LIN {X 120, Y 138, Z 22} c_vel
LIN {X 115, Y 118, Z 22} c_vel
LIN {X 112, Y 106, Z 22} c_vel
LIN {X 111, Y 96, Z 22} c_vel
LIN {X 110, Y 88, Z 22} c_vel
LIN {X 110, Y 81, Z 22} c_vel
LIN {X 111, Y 74, Z 22} c_vel
LIN {X 113, Y 69, Z 22} c_vel
LIN {X 116, Y 63, Z 22} c_vel
LIN {X 119, Y 58, Z 22} c_vel
LIN {X 124, Y 53, Z 22} c_vel
LIN {X 130, Y 48, Z 22} c_vel
LIN {X 138, Y 43, Z 22} c_vel
LIN {X 111, Y 0, Z 22} c_vel
$OUT[4] = FALSE
WAIT SEC 10.0
LIN {X 111, Y 0, Z 23} c_vel
$OUT[4] = TRUE
LIN {X 111, Y 0, Z 23} c_vel
LIN {X 106, Y 3, Z 23} c_vel
LIN {X 97, Y 9, Z 23} c_vel
LIN {X 89, Y 16, Z 23} c_vel
LIN {X 83, Y 23, Z 23} c_vel
LIN {X 77, Y 31, Z 23} c_vel
LIN {X 71, Y 39, Z 23} c_vel
LIN {X 67, Y 47, Z 23} c_vel
LIN {X 64, Y 56, Z 23} c_vel
LIN {X 62, Y 64, Z 23} c_vel
LIN {X 60, Y 73, Z 23} c_vel
LIN {X 59, Y 82, Z 23} c_vel
LIN {X 59, Y 92, Z 23} c_vel
LIN {X 60, Y 103, Z 23} c_vel
LIN {X 62, Y 114, Z 23} c_vel
LIN {X 65, Y 127, Z 23} c_vel
LIN {X 69, Y 144, Z 23} c_vel
LIN {X 74, Y 163, Z 23} c_vel
LIN {X 79, Y 180, Z 23} c_vel
LIN {X 81, Y 191, Z 23} c_vel
LIN {X 82, Y 201, Z 23} c_vel
LIN {X 82, Y 209, Z 23} c_vel
LIN {X 82, Y 217, Z 23} c_vel
LIN {X 80, Y 223, Z 23} c_vel
LIN {X 78, Y 229, Z 23} c_vel
LIN {X 75, Y 234, Z 23} c_vel
LIN {X 71, Y 240, Z 23} c_vel
LIN {X 66, Y 245, Z 23} c_vel
LIN {X 60, Y 250, Z 23} c_vel
LIN {X 52, Y 256, Z 23} c_vel
LIN {X 42, Y 261, Z 23} c_vel
LIN {X 30, Y 267, Z 23} c_vel
LIN {X 16, Y 273, Z 23} c_vel
LIN {X 0, Y 278, Z 23} c_vel
LIN {X 14, Y 327, Z 23} c_vel
LIN {X 28, Y 322, Z 23} c_vel
LIN {X 43, Y 317, Z 23} c_vel
LIN {X 57, Y 311, Z 23} c_vel
LIN {X 70, Y 304, Z 23} c_vel
LIN {X 81, Y 298, Z 23} c_vel
LIN {X 90, Y 291, Z 23} c_vel
LIN {X 99, Y 284, Z 23} c_vel
LIN {X 106, Y 277, Z 23} c_vel
LIN {X 113, Y 269, Z 23} c_vel
LIN {X 118, Y 261, Z 23} c_vel
LIN {X 123, Y 253, Z 23} c_vel
LIN {X 127, Y 244, Z 23} c_vel
LIN {X 130, Y 235, Z 23} c_vel
LIN {X 131, Y 226, Z 23} c_vel
LIN {X 133, Y 217, Z 23} c_vel
LIN {X 133, Y 207, Z 23} c_vel
LIN {X 133, Y 197, Z 23} c_vel
LIN {X 131, Y 186, Z 23} c_vel
LIN {X 129, Y 173, Z 23} c_vel
LIN {X 126, Y 160, Z 23} c_vel
LIN {X 120, Y 138, Z 23} c_vel
LIN {X 115, Y 118, Z 23} c_vel
LIN {X 112, Y 106, Z 23} c_vel
LIN {X 111, Y 96, Z 23} c_vel
LIN {X 110, Y 88, Z 23} c_vel
LIN {X 110, Y 81, Z 23} c_vel
LIN {X 111, Y 74, Z 23} c_vel
LIN {X 113, Y 69, Z 23} c_vel
LIN {X 116, Y 63, Z 23} c_vel
LIN {X 119, Y 58, Z 23} c_vel
LIN {X 124, Y 53, Z 23} c_vel
LIN {X 130, Y 48, Z 23} c_vel
LIN {X 138, Y 43, Z 23} c_vel
LIN {X 111, Y 0, Z 23} c_vel
$OUT[4] = FALSE
WAIT SEC 10.0
LIN {X 111, Y 0, Z 24} c_vel
$OUT[4] = TRUE
LIN {X 111, Y 0, Z 24} c_vel
LIN {X 106, Y 3, Z 24} c_vel
LIN {X 97, Y 9, Z 24} c_vel
LIN {X 89, Y 16, Z 24} c_vel
LIN {X 83, Y 23, Z 24} c_vel
LIN {X 77, Y 31, Z 24} c_vel
LIN {X 71, Y 39, Z 24} c_vel
LIN {X 67, Y 47, Z 24} c_vel
LIN {X 64, Y 56, Z 24} c_vel
LIN {X 62, Y 64, Z 24} c_vel
LIN {X 60, Y 73, Z 24} c_vel
LIN {X 59, Y 82, Z 24} c_vel
LIN {X 59, Y 92, Z 24} c_vel
LIN {X 60, Y 103, Z 24} c_vel
LIN {X 62, Y 114, Z 24} c_vel
LIN {X 65, Y 127, Z 24} c_vel
LIN {X 69, Y 144, Z 24} c_vel
LIN {X 74, Y 163, Z 24} c_vel
LIN {X 79, Y 180, Z 24} c_vel
LIN {X 81, Y 191, Z 24} c_vel
LIN {X 82, Y 201, Z 24} c_vel
LIN {X 82, Y 209, Z 24} c_vel
LIN {X 82, Y 217, Z 24} c_vel
LIN {X 80, Y 223, Z 24} c_vel
LIN {X 78, Y 229, Z 24} c_vel
LIN {X 75, Y 234, Z 24} c_vel
LIN {X 71, Y 240, Z 24} c_vel
LIN {X 66, Y 245, Z 24} c_vel
LIN {X 60, Y 250, Z 24} c_vel
LIN {X 52, Y 256, Z 24} c_vel
LIN {X 42, Y 261, Z 24} c_vel
LIN {X 30, Y 267, Z 24} c_vel
LIN {X 16, Y 273, Z 24} c_vel
LIN {X 0, Y 278, Z 24} c_vel
LIN {X 14, Y 327, Z 24} c_vel
LIN {X 28, Y 322, Z 24} c_vel
LIN {X 43, Y 317, Z 24} c_vel
LIN {X 57, Y 311, Z 24} c_vel
LIN {X 70, Y 304, Z 24} c_vel
LIN {X 81, Y 298, Z 24} c_vel
LIN {X 90, Y 291, Z 24} c_vel
LIN {X 99, Y 284, Z 24} c_vel
LIN {X 106, Y 277, Z 24} c_vel
LIN {X 113, Y 269, Z 24} c_vel
LIN {X 118, Y 261, Z 24} c_vel
LIN {X 123, Y 253, Z 24} c_vel
LIN {X 127, Y 244, Z 24} c_vel
LIN {X 130, Y 235, Z 24} c_vel
LIN {X 131, Y 226, Z 24} c_vel
LIN {X 133, Y 217, Z 24} c_vel
LIN {X 133, Y 207, Z 24} c_vel
LIN {X 133, Y 197, Z 24} c_vel
LIN {X 131, Y 186, Z 24} c_vel
LIN {X 129, Y 173, Z 24} c_vel
LIN {X 126, Y 160, Z 24} c_vel
LIN {X 120, Y 138, Z 24} c_vel
LIN {X 115, Y 118, Z 24} c_vel
LIN {X 112, Y 106, Z 24} c_vel
LIN {X 111, Y 96, Z 24} c_vel
LIN {X 110, Y 88, Z 24} c_vel
LIN {X 110, Y 81, Z 24} c_vel
LIN {X 111, Y 74, Z 24} c_vel
LIN {X 113, Y 69, Z 24} c_vel
LIN {X 116, Y 63, Z 24} c_vel
LIN {X 119, Y 58, Z 24} c_vel
LIN {X 124, Y 53, Z 24} c_vel
LIN {X 130, Y 48, Z 24} c_vel
LIN {X 138, Y 43, Z 24} c_vel
LIN {X 111, Y 0, Z 24} c_vel
$OUT[4] = FALSE
WAIT SEC 10.0
LIN {X 111, Y 0, Z 25} c_vel
$OUT[4] = TRUE
LIN {X 111, Y 0, Z 25} c_vel
LIN {X 106, Y 3, Z 25} c_vel
LIN {X 97, Y 9, Z 25} c_vel
LIN {X 89, Y 16, Z 25} c_vel
LIN {X 83, Y 23, Z 25} c_vel
LIN {X 77, Y 31, Z 25} c_vel
LIN {X 71, Y 39, Z 25} c_vel
LIN {X 67, Y 47, Z 25} c_vel
LIN {X 64, Y 56, Z 25} c_vel
LIN {X 62, Y 64, Z 25} c_vel
LIN {X 60, Y 73, Z 25} c_vel
LIN {X 59, Y 82, Z 25} c_vel
LIN {X 59, Y 92, Z 25} c_vel
LIN {X 60, Y 103, Z 25} c_vel
LIN {X 62, Y 114, Z 25} c_vel
LIN {X 65, Y 127, Z 25} c_vel
LIN {X 69, Y 144, Z 25} c_vel
LIN {X 74, Y 163, Z 25} c_vel
LIN {X 79, Y 180, Z 25} c_vel
LIN {X 81, Y 191, Z 25} c_vel
LIN {X 82, Y 201, Z 25} c_vel
LIN {X 82, Y 209, Z 25} c_vel
LIN {X 82, Y 217, Z 25} c_vel
LIN {X 80, Y 223, Z 25} c_vel
LIN {X 78, Y 229, Z 25} c_vel
LIN {X 75, Y 234, Z 25} c_vel
LIN {X 71, Y 240, Z 25} c_vel
LIN {X 66, Y 245, Z 25} c_vel
LIN {X 60, Y 250, Z 25} c_vel
LIN {X 52, Y 256, Z 25} c_vel
LIN {X 42, Y 261, Z 25} c_vel
LIN {X 30, Y 267, Z 25} c_vel
LIN {X 16, Y 273, Z 25} c_vel
LIN {X 0, Y 278, Z 25} c_vel
LIN {X 14, Y 327, Z 25} c_vel
LIN {X 28, Y 322, Z 25} c_vel
LIN {X 43, Y 317, Z 25} c_vel
LIN {X 57, Y 311, Z 25} c_vel
LIN {X 70, Y 304, Z 25} c_vel
LIN {X 81, Y 298, Z 25} c_vel
LIN {X 90, Y 291, Z 25} c_vel
LIN {X 99, Y 284, Z 25} c_vel
LIN {X 106, Y 277, Z 25} c_vel
LIN {X 113, Y 269, Z 25} c_vel
LIN {X 118, Y 261, Z 25} c_vel
LIN {X 123, Y 253, Z 25} c_vel
LIN {X 127, Y 244, Z 25} c_vel
LIN {X 130, Y 235, Z 25} c_vel
LIN {X 131, Y 226, Z 25} c_vel
LIN {X 133, Y 217, Z 25} c_vel
LIN {X 133, Y 207, Z 25} c_vel
LIN {X 133, Y 197, Z 25} c_vel
LIN {X 131, Y 186, Z 25} c_vel
LIN {X 129, Y 173, Z 25} c_vel
LIN {X 126, Y 160, Z 25} c_vel
LIN {X 120, Y 138, Z 25} c_vel
LIN {X 115, Y 118, Z 25} c_vel
LIN {X 112, Y 106, Z 25} c_vel
LIN {X 111, Y 96, Z 25} c_vel
LIN {X 110, Y 88, Z 25} c_vel
LIN {X 110, Y 81, Z 25} c_vel
LIN {X 111, Y 74, Z 25} c_vel
LIN {X 113, Y 69, Z 25} c_vel
LIN {X 116, Y 63, Z 25} c_vel
LIN {X 119, Y 58, Z 25} c_vel
LIN {X 124, Y 53, Z 25} c_vel
LIN {X 130, Y 48, Z 25} c_vel
LIN {X 138, Y 43, Z 25} c_vel
LIN {X 111, Y 0, Z 25} c_vel
$OUT[4] = FALSE
WAIT SEC 10.0
LIN {X 111, Y 0, Z 26} c_vel
$OUT[4] = TRUE
LIN {X 111, Y 0, Z 26} c_vel
LIN {X 106, Y 3, Z 26} c_vel
LIN {X 97, Y 9, Z 26} c_vel
LIN {X 89, Y 16, Z 26} c_vel
LIN {X 83, Y 23, Z 26} c_vel
LIN {X 77, Y 31, Z 26} c_vel
LIN {X 71, Y 39, Z 26} c_vel
LIN {X 67, Y 47, Z 26} c_vel
LIN {X 64, Y 56, Z 26} c_vel
LIN {X 62, Y 64, Z 26} c_vel
LIN {X 60, Y 73, Z 26} c_vel
LIN {X 59, Y 82, Z 26} c_vel
LIN {X 59, Y 92, Z 26} c_vel
LIN {X 60, Y 103, Z 26} c_vel
LIN {X 62, Y 114, Z 26} c_vel
LIN {X 65, Y 127, Z 26} c_vel
LIN {X 69, Y 144, Z 26} c_vel
LIN {X 74, Y 163, Z 26} c_vel
LIN {X 79, Y 180, Z 26} c_vel
LIN {X 81, Y 191, Z 26} c_vel
LIN {X 82, Y 201, Z 26} c_vel
LIN {X 82, Y 209, Z 26} c_vel
LIN {X 82, Y 217, Z 26} c_vel
LIN {X 80, Y 223, Z 26} c_vel
LIN {X 78, Y 229, Z 26} c_vel
LIN {X 75, Y 234, Z 26} c_vel
LIN {X 71, Y 240, Z 26} c_vel
LIN {X 66, Y 245, Z 26} c_vel
LIN {X 60, Y 250, Z 26} c_vel
LIN {X 52, Y 256, Z 26} c_vel
LIN {X 42, Y 261, Z 26} c_vel
LIN {X 30, Y 267, Z 26} c_vel
LIN {X 16, Y 273, Z 26} c_vel
LIN {X 0, Y 278, Z 26} c_vel
LIN {X 14, Y 327, Z 26} c_vel
LIN {X 28, Y 322, Z 26} c_vel
LIN {X 43, Y 317, Z 26} c_vel
LIN {X 57, Y 311, Z 26} c_vel
LIN {X 70, Y 304, Z 26} c_vel
LIN {X 81, Y 298, Z 26} c_vel
LIN {X 90, Y 291, Z 26} c_vel
LIN {X 99, Y 284, Z 26} c_vel
LIN {X 106, Y 277, Z 26} c_vel
LIN {X 113, Y 269, Z 26} c_vel
LIN {X 118, Y 261, Z 26} c_vel
LIN {X 123, Y 253, Z 26} c_vel
LIN {X 127, Y 244, Z 26} c_vel
LIN {X 130, Y 235, Z 26} c_vel
LIN {X 131, Y 226, Z 26} c_vel
LIN {X 133, Y 217, Z 26} c_vel
LIN {X 133, Y 207, Z 26} c_vel
LIN {X 133, Y 197, Z 26} c_vel
LIN {X 131, Y 186, Z 26} c_vel
LIN {X 129, Y 173, Z 26} c_vel
LIN {X 126, Y 160, Z 26} c_vel
LIN {X 120, Y 138, Z 26} c_vel
LIN {X 115, Y 118, Z 26} c_vel
LIN {X 112, Y 106, Z 26} c_vel
LIN {X 111, Y 96, Z 26} c_vel
LIN {X 110, Y 88, Z 26} c_vel
LIN {X 110, Y 81, Z 26} c_vel
LIN {X 111, Y 74, Z 26} c_vel
LIN {X 113, Y 69, Z 26} c_vel
LIN {X 116, Y 63, Z 26} c_vel
LIN {X 119, Y 58, Z 26} c_vel
LIN {X 124, Y 53, Z 26} c_vel
LIN {X 130, Y 48, Z 26} c_vel
LIN {X 138, Y 43, Z 26} c_vel
LIN {X 111, Y 0, Z 26} c_vel
$OUT[4] = FALSE
WAIT SEC 10.0
LIN {X 111, Y 0, Z 27} c_vel
$OUT[4] = TRUE
LIN {X 111, Y 0, Z 27} c_vel
LIN {X 106, Y 3, Z 27} c_vel
LIN {X 97, Y 9, Z 27} c_vel
LIN {X 89, Y 16, Z 27} c_vel
LIN {X 83, Y 23, Z 27} c_vel
LIN {X 77, Y 31, Z 27} c_vel
LIN {X 71, Y 39, Z 27} c_vel
LIN {X 67, Y 47, Z 27} c_vel
LIN {X 64, Y 56, Z 27} c_vel
LIN {X 62, Y 64, Z 27} c_vel
LIN {X 60, Y 73, Z 27} c_vel
LIN {X 59, Y 82, Z 27} c_vel
LIN {X 59, Y 92, Z 27} c_vel
LIN {X 60, Y 103, Z 27} c_vel
LIN {X 62, Y 114, Z 27} c_vel
LIN {X 65, Y 127, Z 27} c_vel
LIN {X 69, Y 144, Z 27} c_vel
LIN {X 74, Y 163, Z 27} c_vel
LIN {X 79, Y 180, Z 27} c_vel
LIN {X 81, Y 191, Z 27} c_vel
LIN {X 82, Y 201, Z 27} c_vel
LIN {X 82, Y 209, Z 27} c_vel
LIN {X 82, Y 217, Z 27} c_vel
LIN {X 80, Y 223, Z 27} c_vel
LIN {X 78, Y 229, Z 27} c_vel
LIN {X 75, Y 234, Z 27} c_vel
LIN {X 71, Y 240, Z 27} c_vel
LIN {X 66, Y 245, Z 27} c_vel
LIN {X 60, Y 250, Z 27} c_vel
LIN {X 52, Y 256, Z 27} c_vel
LIN {X 42, Y 261, Z 27} c_vel
LIN {X 30, Y 267, Z 27} c_vel
LIN {X 16, Y 273, Z 27} c_vel
LIN {X 0, Y 278, Z 27} c_vel
LIN {X 14, Y 327, Z 27} c_vel
LIN {X 28, Y 322, Z 27} c_vel
LIN {X 43, Y 317, Z 27} c_vel
LIN {X 57, Y 311, Z 27} c_vel
LIN {X 70, Y 304, Z 27} c_vel
LIN {X 81, Y 298, Z 27} c_vel
LIN {X 90, Y 291, Z 27} c_vel
LIN {X 99, Y 284, Z 27} c_vel
LIN {X 106, Y 277, Z 27} c_vel
LIN {X 113, Y 269, Z 27} c_vel
LIN {X 118, Y 261, Z 27} c_vel
LIN {X 123, Y 253, Z 27} c_vel
LIN {X 127, Y 244, Z 27} c_vel
LIN {X 130, Y 235, Z 27} c_vel
LIN {X 131, Y 226, Z 27} c_vel
LIN {X 133, Y 217, Z 27} c_vel
LIN {X 133, Y 207, Z 27} c_vel
LIN {X 133, Y 197, Z 27} c_vel
LIN {X 131, Y 186, Z 27} c_vel
LIN {X 129, Y 173, Z 27} c_vel
LIN {X 126, Y 160, Z 27} c_vel
LIN {X 120, Y 138, Z 27} c_vel
LIN {X 115, Y 118, Z 27} c_vel
LIN {X 112, Y 106, Z 27} c_vel
LIN {X 111, Y 96, Z 27} c_vel
LIN {X 110, Y 88, Z 27} c_vel
LIN {X 110, Y 81, Z 27} c_vel
LIN {X 111, Y 74, Z 27} c_vel
LIN {X 113, Y 69, Z 27} c_vel
LIN {X 116, Y 63, Z 27} c_vel
LIN {X 119, Y 58, Z 27} c_vel
LIN {X 124, Y 53, Z 27} c_vel
LIN {X 130, Y 48, Z 27} c_vel
LIN {X 138, Y 43, Z 27} c_vel
LIN {X 111, Y 0, Z 27} c_vel
$OUT[4] = FALSE
WAIT SEC 10.0
LIN {X 111, Y 0, Z 28} c_vel
$OUT[4] = TRUE
LIN {X 111, Y 0, Z 28} c_vel
LIN {X 106, Y 3, Z 28} c_vel
LIN {X 97, Y 9, Z 28} c_vel
LIN {X 89, Y 16, Z 28} c_vel
LIN {X 83, Y 23, Z 28} c_vel
LIN {X 77, Y 31, Z 28} c_vel
LIN {X 71, Y 39, Z 28} c_vel
LIN {X 67, Y 47, Z 28} c_vel
LIN {X 64, Y 56, Z 28} c_vel
LIN {X 62, Y 64, Z 28} c_vel
LIN {X 60, Y 73, Z 28} c_vel
LIN {X 59, Y 82, Z 28} c_vel
LIN {X 59, Y 92, Z 28} c_vel
LIN {X 60, Y 103, Z 28} c_vel
LIN {X 62, Y 114, Z 28} c_vel
LIN {X 65, Y 127, Z 28} c_vel
LIN {X 69, Y 144, Z 28} c_vel
LIN {X 74, Y 163, Z 28} c_vel
LIN {X 79, Y 180, Z 28} c_vel
LIN {X 81, Y 191, Z 28} c_vel
LIN {X 82, Y 201, Z 28} c_vel
LIN {X 82, Y 209, Z 28} c_vel
LIN {X 82, Y 217, Z 28} c_vel
LIN {X 80, Y 223, Z 28} c_vel
LIN {X 78, Y 229, Z 28} c_vel
LIN {X 75, Y 234, Z 28} c_vel
LIN {X 71, Y 240, Z 28} c_vel
LIN {X 66, Y 245, Z 28} c_vel
LIN {X 60, Y 250, Z 28} c_vel
LIN {X 52, Y 256, Z 28} c_vel
LIN {X 42, Y 261, Z 28} c_vel
LIN {X 30, Y 267, Z 28} c_vel
LIN {X 16, Y 273, Z 28} c_vel
LIN {X 0, Y 278, Z 28} c_vel
LIN {X 14, Y 327, Z 28} c_vel
LIN {X 28, Y 322, Z 28} c_vel
LIN {X 43, Y 317, Z 28} c_vel
LIN {X 57, Y 311, Z 28} c_vel
LIN {X 70, Y 304, Z 28} c_vel
LIN {X 81, Y 298, Z 28} c_vel
LIN {X 90, Y 291, Z 28} c_vel
LIN {X 99, Y 284, Z 28} c_vel
LIN {X 106, Y 277, Z 28} c_vel
LIN {X 113, Y 269, Z 28} c_vel
LIN {X 118, Y 261, Z 28} c_vel
LIN {X 123, Y 253, Z 28} c_vel
LIN {X 127, Y 244, Z 28} c_vel
LIN {X 130, Y 235, Z 28} c_vel
LIN {X 131, Y 226, Z 28} c_vel
LIN {X 133, Y 217, Z 28} c_vel
LIN {X 133, Y 207, Z 28} c_vel
LIN {X 133, Y 197, Z 28} c_vel
LIN {X 131, Y 186, Z 28} c_vel
LIN {X 129, Y 173, Z 28} c_vel
LIN {X 126, Y 160, Z 28} c_vel
LIN {X 120, Y 138, Z 28} c_vel
LIN {X 115, Y 118, Z 28} c_vel
LIN {X 112, Y 106, Z 28} c_vel
LIN {X 111, Y 96, Z 28} c_vel
LIN {X 110, Y 88, Z 28} c_vel
LIN {X 110, Y 81, Z 28} c_vel
LIN {X 111, Y 74, Z 28} c_vel
LIN {X 113, Y 69, Z 28} c_vel
LIN {X 116, Y 63, Z 28} c_vel
LIN {X 119, Y 58, Z 28} c_vel
LIN {X 124, Y 53, Z 28} c_vel
LIN {X 130, Y 48, Z 28} c_vel
LIN {X 138, Y 43, Z 28} c_vel
LIN {X 111, Y 0, Z 28} c_vel
$OUT[4] = FALSE
WAIT SEC 10.0
LIN {X 111, Y 0, Z 29} c_vel
$OUT[4] = TRUE
LIN {X 111, Y 0, Z 29} c_vel
LIN {X 106, Y 3, Z 29} c_vel
LIN {X 97, Y 9, Z 29} c_vel
LIN {X 89, Y 16, Z 29} c_vel
LIN {X 83, Y 23, Z 29} c_vel
LIN {X 77, Y 31, Z 29} c_vel
LIN {X 71, Y 39, Z 29} c_vel
LIN {X 67, Y 47, Z 29} c_vel
LIN {X 64, Y 56, Z 29} c_vel
LIN {X 62, Y 64, Z 29} c_vel
LIN {X 60, Y 73, Z 29} c_vel
LIN {X 59, Y 82, Z 29} c_vel
LIN {X 59, Y 92, Z 29} c_vel
LIN {X 60, Y 103, Z 29} c_vel
LIN {X 62, Y 114, Z 29} c_vel
LIN {X 65, Y 127, Z 29} c_vel
LIN {X 69, Y 144, Z 29} c_vel
LIN {X 74, Y 163, Z 29} c_vel
LIN {X 79, Y 180, Z 29} c_vel
LIN {X 81, Y 191, Z 29} c_vel
LIN {X 82, Y 201, Z 29} c_vel
LIN {X 82, Y 209, Z 29} c_vel
LIN {X 82, Y 217, Z 29} c_vel
LIN {X 80, Y 223, Z 29} c_vel
LIN {X 78, Y 229, Z 29} c_vel
LIN {X 75, Y 234, Z 29} c_vel
LIN {X 71, Y 240, Z 29} c_vel
LIN {X 66, Y 245, Z 29} c_vel
LIN {X 60, Y 250, Z 29} c_vel
LIN {X 52, Y 256, Z 29} c_vel
LIN {X 42, Y 261, Z 29} c_vel
LIN {X 30, Y 267, Z 29} c_vel
LIN {X 16, Y 273, Z 29} c_vel
LIN {X 0, Y 278, Z 29} c_vel
LIN {X 14, Y 327, Z 29} c_vel
LIN {X 28, Y 322, Z 29} c_vel
LIN {X 43, Y 317, Z 29} c_vel
LIN {X 57, Y 311, Z 29} c_vel
LIN {X 70, Y 304, Z 29} c_vel
LIN {X 81, Y 298, Z 29} c_vel
LIN {X 90, Y 291, Z 29} c_vel
LIN {X 99, Y 284, Z 29} c_vel
LIN {X 106, Y 277, Z 29} c_vel
LIN {X 113, Y 269, Z 29} c_vel
LIN {X 118, Y 261, Z 29} c_vel
LIN {X 123, Y 253, Z 29} c_vel
LIN {X 127, Y 244, Z 29} c_vel
LIN {X 130, Y 235, Z 29} c_vel
LIN {X 131, Y 226, Z 29} c_vel
LIN {X 133, Y 217, Z 29} c_vel
LIN {X 133, Y 207, Z 29} c_vel
LIN {X 133, Y 197, Z 29} c_vel
LIN {X 131, Y 186, Z 29} c_vel
LIN {X 129, Y 173, Z 29} c_vel
LIN {X 126, Y 160, Z 29} c_vel
LIN {X 120, Y 138, Z 29} c_vel
LIN {X 115, Y 118, Z 29} c_vel
LIN {X 112, Y 106, Z 29} c_vel
LIN {X 111, Y 96, Z 29} c_vel
LIN {X 110, Y 88, Z 29} c_vel
LIN {X 110, Y 81, Z 29} c_vel
LIN {X 111, Y 74, Z 29} c_vel
LIN {X 113, Y 69, Z 29} c_vel
LIN {X 116, Y 63, Z 29} c_vel
LIN {X 119, Y 58, Z 29} c_vel
LIN {X 124, Y 53, Z 29} c_vel
LIN {X 130, Y 48, Z 29} c_vel
LIN {X 138, Y 43, Z 29} c_vel
LIN {X 111, Y 0, Z 29} c_vel
$OUT[4] = FALSE
WAIT SEC 10.0
LIN {X 111, Y 0, Z 30} c_vel
$OUT[4] = TRUE
LIN {X 111, Y 0, Z 30} c_vel
LIN {X 106, Y 3, Z 30} c_vel
LIN {X 97, Y 9, Z 30} c_vel
LIN {X 89, Y 16, Z 30} c_vel
LIN {X 83, Y 23, Z 30} c_vel
LIN {X 77, Y 31, Z 30} c_vel
LIN {X 71, Y 39, Z 30} c_vel
LIN {X 67, Y 47, Z 30} c_vel
LIN {X 64, Y 56, Z 30} c_vel
LIN {X 62, Y 64, Z 30} c_vel
LIN {X 60, Y 73, Z 30} c_vel
LIN {X 59, Y 82, Z 30} c_vel
LIN {X 59, Y 92, Z 30} c_vel
LIN {X 60, Y 103, Z 30} c_vel
LIN {X 62, Y 114, Z 30} c_vel
LIN {X 65, Y 127, Z 30} c_vel
LIN {X 69, Y 144, Z 30} c_vel
LIN {X 74, Y 163, Z 30} c_vel
LIN {X 79, Y 180, Z 30} c_vel
LIN {X 81, Y 191, Z 30} c_vel
LIN {X 82, Y 201, Z 30} c_vel
LIN {X 82, Y 209, Z 30} c_vel
LIN {X 82, Y 217, Z 30} c_vel
LIN {X 80, Y 223, Z 30} c_vel
LIN {X 78, Y 229, Z 30} c_vel
LIN {X 75, Y 234, Z 30} c_vel
LIN {X 71, Y 240, Z 30} c_vel
LIN {X 66, Y 245, Z 30} c_vel
LIN {X 60, Y 250, Z 30} c_vel
LIN {X 52, Y 256, Z 30} c_vel
LIN {X 42, Y 261, Z 30} c_vel
LIN {X 30, Y 267, Z 30} c_vel
LIN {X 16, Y 273, Z 30} c_vel
LIN {X 0, Y 278, Z 30} c_vel
LIN {X 14, Y 327, Z 30} c_vel
LIN {X 28, Y 322, Z 30} c_vel
LIN {X 43, Y 317, Z 30} c_vel
LIN {X 57, Y 311, Z 30} c_vel
LIN {X 70, Y 304, Z 30} c_vel
LIN {X 81, Y 298, Z 30} c_vel
LIN {X 90, Y 291, Z 30} c_vel
LIN {X 99, Y 284, Z 30} c_vel
LIN {X 106, Y 277, Z 30} c_vel
LIN {X 113, Y 269, Z 30} c_vel
LIN {X 118, Y 261, Z 30} c_vel
LIN {X 123, Y 253, Z 30} c_vel
LIN {X 127, Y 244, Z 30} c_vel
LIN {X 130, Y 235, Z 30} c_vel
LIN {X 131, Y 226, Z 30} c_vel
LIN {X 133, Y 217, Z 30} c_vel
LIN {X 133, Y 207, Z 30} c_vel
LIN {X 133, Y 197, Z 30} c_vel
LIN {X 131, Y 186, Z 30} c_vel
LIN {X 129, Y 173, Z 30} c_vel
LIN {X 126, Y 160, Z 30} c_vel
LIN {X 120, Y 138, Z 30} c_vel
LIN {X 115, Y 118, Z 30} c_vel
LIN {X 112, Y 106, Z 30} c_vel
LIN {X 111, Y 96, Z 30} c_vel
LIN {X 110, Y 88, Z 30} c_vel
LIN {X 110, Y 81, Z 30} c_vel
LIN {X 111, Y 74, Z 30} c_vel
LIN {X 113, Y 69, Z 30} c_vel
LIN {X 116, Y 63, Z 30} c_vel
LIN {X 119, Y 58, Z 30} c_vel
LIN {X 124, Y 53, Z 30} c_vel
LIN {X 130, Y 48, Z 30} c_vel
LIN {X 138, Y 43, Z 30} c_vel
LIN {X 111, Y 0, Z 30} c_vel
$OUT[4] = FALSE
WAIT SEC 10.0
LIN {X 111, Y 0, Z 31} c_vel
$OUT[4] = TRUE
LIN {X 111, Y 0, Z 31} c_vel
LIN {X 106, Y 3, Z 31} c_vel
LIN {X 97, Y 9, Z 31} c_vel
LIN {X 89, Y 16, Z 31} c_vel
LIN {X 83, Y 23, Z 31} c_vel
LIN {X 77, Y 31, Z 31} c_vel
LIN {X 71, Y 39, Z 31} c_vel
LIN {X 67, Y 47, Z 31} c_vel
LIN {X 64, Y 56, Z 31} c_vel
LIN {X 62, Y 64, Z 31} c_vel
LIN {X 60, Y 73, Z 31} c_vel
LIN {X 59, Y 82, Z 31} c_vel
LIN {X 59, Y 92, Z 31} c_vel
LIN {X 60, Y 103, Z 31} c_vel
LIN {X 62, Y 114, Z 31} c_vel
LIN {X 65, Y 127, Z 31} c_vel
LIN {X 69, Y 144, Z 31} c_vel
LIN {X 74, Y 163, Z 31} c_vel
LIN {X 79, Y 180, Z 31} c_vel
LIN {X 81, Y 191, Z 31} c_vel
LIN {X 82, Y 201, Z 31} c_vel
LIN {X 82, Y 209, Z 31} c_vel
LIN {X 82, Y 217, Z 31} c_vel
LIN {X 80, Y 223, Z 31} c_vel
LIN {X 78, Y 229, Z 31} c_vel
LIN {X 75, Y 234, Z 31} c_vel
LIN {X 71, Y 240, Z 31} c_vel
LIN {X 66, Y 245, Z 31} c_vel
LIN {X 60, Y 250, Z 31} c_vel
LIN {X 52, Y 256, Z 31} c_vel
LIN {X 42, Y 261, Z 31} c_vel
LIN {X 30, Y 267, Z 31} c_vel
LIN {X 16, Y 273, Z 31} c_vel
LIN {X 0, Y 278, Z 31} c_vel
LIN {X 14, Y 327, Z 31} c_vel
LIN {X 28, Y 322, Z 31} c_vel
LIN {X 43, Y 317, Z 31} c_vel
LIN {X 57, Y 311, Z 31} c_vel
LIN {X 70, Y 304, Z 31} c_vel
LIN {X 81, Y 298, Z 31} c_vel
LIN {X 90, Y 291, Z 31} c_vel
LIN {X 99, Y 284, Z 31} c_vel
LIN {X 106, Y 277, Z 31} c_vel
LIN {X 113, Y 269, Z 31} c_vel
LIN {X 118, Y 261, Z 31} c_vel
LIN {X 123, Y 253, Z 31} c_vel
LIN {X 127, Y 244, Z 31} c_vel
LIN {X 130, Y 235, Z 31} c_vel
LIN {X 131, Y 226, Z 31} c_vel
LIN {X 133, Y 217, Z 31} c_vel
LIN {X 133, Y 207, Z 31} c_vel
LIN {X 133, Y 197, Z 31} c_vel
LIN {X 131, Y 186, Z 31} c_vel
LIN {X 129, Y 173, Z 31} c_vel
LIN {X 126, Y 160, Z 31} c_vel
LIN {X 120, Y 138, Z 31} c_vel
LIN {X 115, Y 118, Z 31} c_vel
LIN {X 112, Y 106, Z 31} c_vel
LIN {X 111, Y 96, Z 31} c_vel
LIN {X 110, Y 88, Z 31} c_vel
LIN {X 110, Y 81, Z 31} c_vel
LIN {X 111, Y 74, Z 31} c_vel
LIN {X 113, Y 69, Z 31} c_vel
LIN {X 116, Y 63, Z 31} c_vel
LIN {X 119, Y 58, Z 31} c_vel
LIN {X 124, Y 53, Z 31} c_vel
LIN {X 130, Y 48, Z 31} c_vel
LIN {X 138, Y 43, Z 31} c_vel
LIN {X 111, Y 0, Z 31} c_vel
$OUT[4] = FALSE
WAIT SEC 10.0
LIN {X 111, Y 0, Z 32} c_vel
$OUT[4] = TRUE
LIN {X 111, Y 0, Z 32} c_vel
LIN {X 106, Y 3, Z 32} c_vel
LIN {X 97, Y 9, Z 32} c_vel
LIN {X 89, Y 16, Z 32} c_vel
LIN {X 83, Y 23, Z 32} c_vel
LIN {X 77, Y 31, Z 32} c_vel
LIN {X 71, Y 39, Z 32} c_vel
LIN {X 67, Y 47, Z 32} c_vel
LIN {X 64, Y 56, Z 32} c_vel
LIN {X 62, Y 64, Z 32} c_vel
LIN {X 60, Y 73, Z 32} c_vel
LIN {X 59, Y 82, Z 32} c_vel
LIN {X 59, Y 92, Z 32} c_vel
LIN {X 60, Y 103, Z 32} c_vel
LIN {X 62, Y 114, Z 32} c_vel
LIN {X 65, Y 127, Z 32} c_vel
LIN {X 69, Y 144, Z 32} c_vel
LIN {X 74, Y 163, Z 32} c_vel
LIN {X 79, Y 180, Z 32} c_vel
LIN {X 81, Y 191, Z 32} c_vel
LIN {X 82, Y 201, Z 32} c_vel
LIN {X 82, Y 209, Z 32} c_vel
LIN {X 82, Y 217, Z 32} c_vel
LIN {X 80, Y 223, Z 32} c_vel
LIN {X 78, Y 229, Z 32} c_vel
LIN {X 75, Y 234, Z 32} c_vel
LIN {X 71, Y 240, Z 32} c_vel
LIN {X 66, Y 245, Z 32} c_vel
LIN {X 60, Y 250, Z 32} c_vel
LIN {X 52, Y 256, Z 32} c_vel
LIN {X 42, Y 261, Z 32} c_vel
LIN {X 30, Y 267, Z 32} c_vel
LIN {X 16, Y 273, Z 32} c_vel
LIN {X 0, Y 278, Z 32} c_vel
LIN {X 14, Y 327, Z 32} c_vel
LIN {X 28, Y 322, Z 32} c_vel
LIN {X 43, Y 317, Z 32} c_vel
LIN {X 57, Y 311, Z 32} c_vel
LIN {X 70, Y 304, Z 32} c_vel
LIN {X 81, Y 298, Z 32} c_vel
LIN {X 90, Y 291, Z 32} c_vel
LIN {X 99, Y 284, Z 32} c_vel
LIN {X 106, Y 277, Z 32} c_vel
LIN {X 113, Y 269, Z 32} c_vel
LIN {X 118, Y 261, Z 32} c_vel
LIN {X 123, Y 253, Z 32} c_vel
LIN {X 127, Y 244, Z 32} c_vel
LIN {X 130, Y 235, Z 32} c_vel
LIN {X 131, Y 226, Z 32} c_vel
LIN {X 133, Y 217, Z 32} c_vel
LIN {X 133, Y 207, Z 32} c_vel
LIN {X 133, Y 197, Z 32} c_vel
LIN {X 131, Y 186, Z 32} c_vel
LIN {X 129, Y 173, Z 32} c_vel
LIN {X 126, Y 160, Z 32} c_vel
LIN {X 120, Y 138, Z 32} c_vel
LIN {X 115, Y 118, Z 32} c_vel
LIN {X 112, Y 106, Z 32} c_vel
LIN {X 111, Y 96, Z 32} c_vel
LIN {X 110, Y 88, Z 32} c_vel
LIN {X 110, Y 81, Z 32} c_vel
LIN {X 111, Y 74, Z 32} c_vel
LIN {X 113, Y 69, Z 32} c_vel
LIN {X 116, Y 63, Z 32} c_vel
LIN {X 119, Y 58, Z 32} c_vel
LIN {X 124, Y 53, Z 32} c_vel
LIN {X 130, Y 48, Z 32} c_vel
LIN {X 138, Y 43, Z 32} c_vel
LIN {X 111, Y 0, Z 32} c_vel
$OUT[4] = FALSE
WAIT SEC 10.0
LIN {X 111, Y 0, Z 33} c_vel
$OUT[4] = TRUE
LIN {X 111, Y 0, Z 33} c_vel
LIN {X 106, Y 3, Z 33} c_vel
LIN {X 97, Y 9, Z 33} c_vel
LIN {X 89, Y 16, Z 33} c_vel
LIN {X 83, Y 23, Z 33} c_vel
LIN {X 77, Y 31, Z 33} c_vel
LIN {X 71, Y 39, Z 33} c_vel
LIN {X 67, Y 47, Z 33} c_vel
LIN {X 64, Y 56, Z 33} c_vel
LIN {X 62, Y 64, Z 33} c_vel
LIN {X 60, Y 73, Z 33} c_vel
LIN {X 59, Y 82, Z 33} c_vel
LIN {X 59, Y 92, Z 33} c_vel
LIN {X 60, Y 103, Z 33} c_vel
LIN {X 62, Y 114, Z 33} c_vel
LIN {X 65, Y 127, Z 33} c_vel
LIN {X 69, Y 144, Z 33} c_vel
LIN {X 74, Y 163, Z 33} c_vel
LIN {X 79, Y 180, Z 33} c_vel
LIN {X 81, Y 191, Z 33} c_vel
LIN {X 82, Y 201, Z 33} c_vel
LIN {X 82, Y 209, Z 33} c_vel
LIN {X 82, Y 217, Z 33} c_vel
LIN {X 80, Y 223, Z 33} c_vel
LIN {X 78, Y 229, Z 33} c_vel
LIN {X 75, Y 234, Z 33} c_vel
LIN {X 71, Y 240, Z 33} c_vel
LIN {X 66, Y 245, Z 33} c_vel
LIN {X 60, Y 250, Z 33} c_vel
LIN {X 52, Y 256, Z 33} c_vel
LIN {X 42, Y 261, Z 33} c_vel
LIN {X 30, Y 267, Z 33} c_vel
LIN {X 16, Y 273, Z 33} c_vel
LIN {X 0, Y 278, Z 33} c_vel
LIN {X 14, Y 327, Z 33} c_vel
LIN {X 28, Y 322, Z 33} c_vel
LIN {X 43, Y 317, Z 33} c_vel
LIN {X 57, Y 311, Z 33} c_vel
LIN {X 70, Y 304, Z 33} c_vel
LIN {X 81, Y 298, Z 33} c_vel
LIN {X 90, Y 291, Z 33} c_vel
LIN {X 99, Y 284, Z 33} c_vel
LIN {X 106, Y 277, Z 33} c_vel
LIN {X 113, Y 269, Z 33} c_vel
LIN {X 118, Y 261, Z 33} c_vel
LIN {X 123, Y 253, Z 33} c_vel
LIN {X 127, Y 244, Z 33} c_vel
LIN {X 130, Y 235, Z 33} c_vel
LIN {X 131, Y 226, Z 33} c_vel
LIN {X 133, Y 217, Z 33} c_vel
LIN {X 133, Y 207, Z 33} c_vel
LIN {X 133, Y 197, Z 33} c_vel
LIN {X 131, Y 186, Z 33} c_vel
LIN {X 129, Y 173, Z 33} c_vel
LIN {X 126, Y 160, Z 33} c_vel
LIN {X 120, Y 138, Z 33} c_vel
LIN {X 115, Y 118, Z 33} c_vel
LIN {X 112, Y 106, Z 33} c_vel
LIN {X 111, Y 96, Z 33} c_vel
LIN {X 110, Y 88, Z 33} c_vel
LIN {X 110, Y 81, Z 33} c_vel
LIN {X 111, Y 74, Z 33} c_vel
LIN {X 113, Y 69, Z 33} c_vel
LIN {X 116, Y 63, Z 33} c_vel
LIN {X 119, Y 58, Z 33} c_vel
LIN {X 124, Y 53, Z 33} c_vel
LIN {X 130, Y 48, Z 33} c_vel
LIN {X 138, Y 43, Z 33} c_vel
LIN {X 111, Y 0, Z 33} c_vel
$OUT[4] = FALSE
WAIT SEC 10.0
LIN {X 111, Y 0, Z 34} c_vel
$OUT[4] = TRUE
LIN {X 111, Y 0, Z 34} c_vel
LIN {X 106, Y 3, Z 34} c_vel
LIN {X 97, Y 9, Z 34} c_vel
LIN {X 89, Y 16, Z 34} c_vel
LIN {X 83, Y 23, Z 34} c_vel
LIN {X 77, Y 31, Z 34} c_vel
LIN {X 71, Y 39, Z 34} c_vel
LIN {X 67, Y 47, Z 34} c_vel
LIN {X 64, Y 56, Z 34} c_vel
LIN {X 62, Y 64, Z 34} c_vel
LIN {X 60, Y 73, Z 34} c_vel
LIN {X 59, Y 82, Z 34} c_vel
LIN {X 59, Y 92, Z 34} c_vel
LIN {X 60, Y 103, Z 34} c_vel
LIN {X 62, Y 114, Z 34} c_vel
LIN {X 65, Y 127, Z 34} c_vel
LIN {X 69, Y 144, Z 34} c_vel
LIN {X 74, Y 163, Z 34} c_vel
LIN {X 79, Y 180, Z 34} c_vel
LIN {X 81, Y 191, Z 34} c_vel
LIN {X 82, Y 201, Z 34} c_vel
LIN {X 82, Y 209, Z 34} c_vel
LIN {X 82, Y 217, Z 34} c_vel
LIN {X 80, Y 223, Z 34} c_vel
LIN {X 78, Y 229, Z 34} c_vel
LIN {X 75, Y 234, Z 34} c_vel
LIN {X 71, Y 240, Z 34} c_vel
LIN {X 66, Y 245, Z 34} c_vel
LIN {X 60, Y 250, Z 34} c_vel
LIN {X 52, Y 256, Z 34} c_vel
LIN {X 42, Y 261, Z 34} c_vel
LIN {X 30, Y 267, Z 34} c_vel
LIN {X 16, Y 273, Z 34} c_vel
LIN {X 0, Y 278, Z 34} c_vel
LIN {X 14, Y 327, Z 34} c_vel
LIN {X 28, Y 322, Z 34} c_vel
LIN {X 43, Y 317, Z 34} c_vel
LIN {X 57, Y 311, Z 34} c_vel
LIN {X 70, Y 304, Z 34} c_vel
LIN {X 81, Y 298, Z 34} c_vel
LIN {X 90, Y 291, Z 34} c_vel
LIN {X 99, Y 284, Z 34} c_vel
LIN {X 106, Y 277, Z 34} c_vel
LIN {X 113, Y 269, Z 34} c_vel
LIN {X 118, Y 261, Z 34} c_vel
LIN {X 123, Y 253, Z 34} c_vel
LIN {X 127, Y 244, Z 34} c_vel
LIN {X 130, Y 235, Z 34} c_vel
LIN {X 131, Y 226, Z 34} c_vel
LIN {X 133, Y 217, Z 34} c_vel
LIN {X 133, Y 207, Z 34} c_vel
LIN {X 133, Y 197, Z 34} c_vel
LIN {X 131, Y 186, Z 34} c_vel
LIN {X 129, Y 173, Z 34} c_vel
LIN {X 126, Y 160, Z 34} c_vel
LIN {X 120, Y 138, Z 34} c_vel
LIN {X 115, Y 118, Z 34} c_vel
LIN {X 112, Y 106, Z 34} c_vel
LIN {X 111, Y 96, Z 34} c_vel
LIN {X 110, Y 88, Z 34} c_vel
LIN {X 110, Y 81, Z 34} c_vel
LIN {X 111, Y 74, Z 34} c_vel
LIN {X 113, Y 69, Z 34} c_vel
LIN {X 116, Y 63, Z 34} c_vel
LIN {X 119, Y 58, Z 34} c_vel
LIN {X 124, Y 53, Z 34} c_vel
LIN {X 130, Y 48, Z 34} c_vel
LIN {X 138, Y 43, Z 34} c_vel
LIN {X 111, Y 0, Z 34} c_vel
$OUT[4] = FALSE
WAIT SEC 10.0
LIN {X 111, Y 0, Z 35} c_vel
$OUT[4] = TRUE
LIN {X 111, Y 0, Z 35} c_vel
LIN {X 106, Y 3, Z 35} c_vel
LIN {X 97, Y 9, Z 35} c_vel
LIN {X 89, Y 16, Z 35} c_vel
LIN {X 83, Y 23, Z 35} c_vel
LIN {X 77, Y 31, Z 35} c_vel
LIN {X 71, Y 39, Z 35} c_vel
LIN {X 67, Y 47, Z 35} c_vel
LIN {X 64, Y 56, Z 35} c_vel
LIN {X 62, Y 64, Z 35} c_vel
LIN {X 60, Y 73, Z 35} c_vel
LIN {X 59, Y 82, Z 35} c_vel
LIN {X 59, Y 92, Z 35} c_vel
LIN {X 60, Y 103, Z 35} c_vel
LIN {X 62, Y 114, Z 35} c_vel
LIN {X 65, Y 127, Z 35} c_vel
LIN {X 69, Y 144, Z 35} c_vel
LIN {X 74, Y 163, Z 35} c_vel
LIN {X 79, Y 180, Z 35} c_vel
LIN {X 81, Y 191, Z 35} c_vel
LIN {X 82, Y 201, Z 35} c_vel
LIN {X 82, Y 209, Z 35} c_vel
LIN {X 82, Y 217, Z 35} c_vel
LIN {X 80, Y 223, Z 35} c_vel
LIN {X 78, Y 229, Z 35} c_vel
LIN {X 75, Y 234, Z 35} c_vel
LIN {X 71, Y 240, Z 35} c_vel
LIN {X 66, Y 245, Z 35} c_vel
LIN {X 60, Y 250, Z 35} c_vel
LIN {X 52, Y 256, Z 35} c_vel
LIN {X 42, Y 261, Z 35} c_vel
LIN {X 30, Y 267, Z 35} c_vel
LIN {X 16, Y 273, Z 35} c_vel
LIN {X 0, Y 278, Z 35} c_vel
LIN {X 14, Y 327, Z 35} c_vel
LIN {X 28, Y 322, Z 35} c_vel
LIN {X 43, Y 317, Z 35} c_vel
LIN {X 57, Y 311, Z 35} c_vel
LIN {X 70, Y 304, Z 35} c_vel
LIN {X 81, Y 298, Z 35} c_vel
LIN {X 90, Y 291, Z 35} c_vel
LIN {X 99, Y 284, Z 35} c_vel
LIN {X 106, Y 277, Z 35} c_vel
LIN {X 113, Y 269, Z 35} c_vel
LIN {X 118, Y 261, Z 35} c_vel
LIN {X 123, Y 253, Z 35} c_vel
LIN {X 127, Y 244, Z 35} c_vel
LIN {X 130, Y 235, Z 35} c_vel
LIN {X 131, Y 226, Z 35} c_vel
LIN {X 133, Y 217, Z 35} c_vel
LIN {X 133, Y 207, Z 35} c_vel
LIN {X 133, Y 197, Z 35} c_vel
LIN {X 131, Y 186, Z 35} c_vel
LIN {X 129, Y 173, Z 35} c_vel
LIN {X 126, Y 160, Z 35} c_vel
LIN {X 120, Y 138, Z 35} c_vel
LIN {X 115, Y 118, Z 35} c_vel
LIN {X 112, Y 106, Z 35} c_vel
LIN {X 111, Y 96, Z 35} c_vel
LIN {X 110, Y 88, Z 35} c_vel
LIN {X 110, Y 81, Z 35} c_vel
LIN {X 111, Y 74, Z 35} c_vel
LIN {X 113, Y 69, Z 35} c_vel
LIN {X 116, Y 63, Z 35} c_vel
LIN {X 119, Y 58, Z 35} c_vel
LIN {X 124, Y 53, Z 35} c_vel
LIN {X 130, Y 48, Z 35} c_vel
LIN {X 138, Y 43, Z 35} c_vel
LIN {X 111, Y 0, Z 35} c_vel
$OUT[4] = FALSE
WAIT SEC 10.0
LIN {X 111, Y 0, Z 36} c_vel
$OUT[4] = TRUE
LIN {X 111, Y 0, Z 36} c_vel
LIN {X 106, Y 3, Z 36} c_vel
LIN {X 97, Y 9, Z 36} c_vel
LIN {X 89, Y 16, Z 36} c_vel
LIN {X 83, Y 23, Z 36} c_vel
LIN {X 77, Y 31, Z 36} c_vel
LIN {X 71, Y 39, Z 36} c_vel
LIN {X 67, Y 47, Z 36} c_vel
LIN {X 64, Y 56, Z 36} c_vel
LIN {X 62, Y 64, Z 36} c_vel
LIN {X 60, Y 73, Z 36} c_vel
LIN {X 59, Y 82, Z 36} c_vel
LIN {X 59, Y 92, Z 36} c_vel
LIN {X 60, Y 103, Z 36} c_vel
LIN {X 62, Y 114, Z 36} c_vel
LIN {X 65, Y 127, Z 36} c_vel
LIN {X 69, Y 144, Z 36} c_vel
LIN {X 74, Y 163, Z 36} c_vel
LIN {X 79, Y 180, Z 36} c_vel
LIN {X 81, Y 191, Z 36} c_vel
LIN {X 82, Y 201, Z 36} c_vel
LIN {X 82, Y 209, Z 36} c_vel
LIN {X 82, Y 217, Z 36} c_vel
LIN {X 80, Y 223, Z 36} c_vel
LIN {X 78, Y 229, Z 36} c_vel
LIN {X 75, Y 234, Z 36} c_vel
LIN {X 71, Y 240, Z 36} c_vel
LIN {X 66, Y 245, Z 36} c_vel
LIN {X 60, Y 250, Z 36} c_vel
LIN {X 52, Y 256, Z 36} c_vel
LIN {X 42, Y 261, Z 36} c_vel
LIN {X 30, Y 267, Z 36} c_vel
LIN {X 16, Y 273, Z 36} c_vel
LIN {X 0, Y 278, Z 36} c_vel
LIN {X 14, Y 327, Z 36} c_vel
LIN {X 28, Y 322, Z 36} c_vel
LIN {X 43, Y 317, Z 36} c_vel
LIN {X 57, Y 311, Z 36} c_vel
LIN {X 70, Y 304, Z 36} c_vel
LIN {X 81, Y 298, Z 36} c_vel
LIN {X 90, Y 291, Z 36} c_vel
LIN {X 99, Y 284, Z 36} c_vel
LIN {X 106, Y 277, Z 36} c_vel
LIN {X 113, Y 269, Z 36} c_vel
LIN {X 118, Y 261, Z 36} c_vel
LIN {X 123, Y 253, Z 36} c_vel
LIN {X 127, Y 244, Z 36} c_vel
LIN {X 130, Y 235, Z 36} c_vel
LIN {X 131, Y 226, Z 36} c_vel
LIN {X 133, Y 217, Z 36} c_vel
LIN {X 133, Y 207, Z 36} c_vel
LIN {X 133, Y 197, Z 36} c_vel
LIN {X 131, Y 186, Z 36} c_vel
LIN {X 129, Y 173, Z 36} c_vel
LIN {X 126, Y 160, Z 36} c_vel
LIN {X 120, Y 138, Z 36} c_vel
LIN {X 115, Y 118, Z 36} c_vel
LIN {X 112, Y 106, Z 36} c_vel
LIN {X 111, Y 96, Z 36} c_vel
LIN {X 110, Y 88, Z 36} c_vel
LIN {X 110, Y 81, Z 36} c_vel
LIN {X 111, Y 74, Z 36} c_vel
LIN {X 113, Y 69, Z 36} c_vel
LIN {X 116, Y 63, Z 36} c_vel
LIN {X 119, Y 58, Z 36} c_vel
LIN {X 124, Y 53, Z 36} c_vel
LIN {X 130, Y 48, Z 36} c_vel
LIN {X 138, Y 43, Z 36} c_vel
LIN {X 111, Y 0, Z 36} c_vel
$OUT[4] = FALSE
WAIT SEC 10.0
LIN {X 111, Y 0, Z 37} c_vel
$OUT[4] = TRUE
LIN {X 111, Y 0, Z 37} c_vel
LIN {X 106, Y 3, Z 37} c_vel
LIN {X 97, Y 9, Z 37} c_vel
LIN {X 89, Y 16, Z 37} c_vel
LIN {X 83, Y 23, Z 37} c_vel
LIN {X 77, Y 31, Z 37} c_vel
LIN {X 71, Y 39, Z 37} c_vel
LIN {X 67, Y 47, Z 37} c_vel
LIN {X 64, Y 56, Z 37} c_vel
LIN {X 62, Y 64, Z 37} c_vel
LIN {X 60, Y 73, Z 37} c_vel
LIN {X 59, Y 82, Z 37} c_vel
LIN {X 59, Y 92, Z 37} c_vel
LIN {X 60, Y 103, Z 37} c_vel
LIN {X 62, Y 114, Z 37} c_vel
LIN {X 65, Y 127, Z 37} c_vel
LIN {X 69, Y 144, Z 37} c_vel
LIN {X 74, Y 163, Z 37} c_vel
LIN {X 79, Y 180, Z 37} c_vel
LIN {X 81, Y 191, Z 37} c_vel
LIN {X 82, Y 201, Z 37} c_vel
LIN {X 82, Y 209, Z 37} c_vel
LIN {X 82, Y 217, Z 37} c_vel
LIN {X 80, Y 223, Z 37} c_vel
LIN {X 78, Y 229, Z 37} c_vel
LIN {X 75, Y 234, Z 37} c_vel
LIN {X 71, Y 240, Z 37} c_vel
LIN {X 66, Y 245, Z 37} c_vel
LIN {X 60, Y 250, Z 37} c_vel
LIN {X 52, Y 256, Z 37} c_vel
LIN {X 42, Y 261, Z 37} c_vel
LIN {X 30, Y 267, Z 37} c_vel
LIN {X 16, Y 273, Z 37} c_vel
LIN {X 0, Y 278, Z 37} c_vel
LIN {X 14, Y 327, Z 37} c_vel
LIN {X 28, Y 322, Z 37} c_vel
LIN {X 43, Y 317, Z 37} c_vel
LIN {X 57, Y 311, Z 37} c_vel
LIN {X 70, Y 304, Z 37} c_vel
LIN {X 81, Y 298, Z 37} c_vel
LIN {X 90, Y 291, Z 37} c_vel
LIN {X 99, Y 284, Z 37} c_vel
LIN {X 106, Y 277, Z 37} c_vel
LIN {X 113, Y 269, Z 37} c_vel
LIN {X 118, Y 261, Z 37} c_vel
LIN {X 123, Y 253, Z 37} c_vel
LIN {X 127, Y 244, Z 37} c_vel
LIN {X 130, Y 235, Z 37} c_vel
LIN {X 131, Y 226, Z 37} c_vel
LIN {X 133, Y 217, Z 37} c_vel
LIN {X 133, Y 207, Z 37} c_vel
LIN {X 133, Y 197, Z 37} c_vel
LIN {X 131, Y 186, Z 37} c_vel
LIN {X 129, Y 173, Z 37} c_vel
LIN {X 126, Y 160, Z 37} c_vel
LIN {X 120, Y 138, Z 37} c_vel
LIN {X 115, Y 118, Z 37} c_vel
LIN {X 112, Y 106, Z 37} c_vel
LIN {X 111, Y 96, Z 37} c_vel
LIN {X 110, Y 88, Z 37} c_vel
LIN {X 110, Y 81, Z 37} c_vel
LIN {X 111, Y 74, Z 37} c_vel
LIN {X 113, Y 69, Z 37} c_vel
LIN {X 116, Y 63, Z 37} c_vel
LIN {X 119, Y 58, Z 37} c_vel
LIN {X 124, Y 53, Z 37} c_vel
LIN {X 130, Y 48, Z 37} c_vel
LIN {X 138, Y 43, Z 37} c_vel
LIN {X 111, Y 0, Z 37} c_vel
$OUT[4] = FALSE
WAIT SEC 10.0
LIN {X 111, Y 0, Z 38} c_vel
$OUT[4] = TRUE
LIN {X 111, Y 0, Z 38} c_vel
LIN {X 106, Y 3, Z 38} c_vel
LIN {X 97, Y 9, Z 38} c_vel
LIN {X 89, Y 16, Z 38} c_vel
LIN {X 83, Y 23, Z 38} c_vel
LIN {X 77, Y 31, Z 38} c_vel
LIN {X 71, Y 39, Z 38} c_vel
LIN {X 67, Y 47, Z 38} c_vel
LIN {X 64, Y 56, Z 38} c_vel
LIN {X 62, Y 64, Z 38} c_vel
LIN {X 60, Y 73, Z 38} c_vel
LIN {X 59, Y 82, Z 38} c_vel
LIN {X 59, Y 92, Z 38} c_vel
LIN {X 60, Y 103, Z 38} c_vel
LIN {X 62, Y 114, Z 38} c_vel
LIN {X 65, Y 127, Z 38} c_vel
LIN {X 69, Y 144, Z 38} c_vel
LIN {X 74, Y 163, Z 38} c_vel
LIN {X 79, Y 180, Z 38} c_vel
LIN {X 81, Y 191, Z 38} c_vel
LIN {X 82, Y 201, Z 38} c_vel
LIN {X 82, Y 209, Z 38} c_vel
LIN {X 82, Y 217, Z 38} c_vel
LIN {X 80, Y 223, Z 38} c_vel
LIN {X 78, Y 229, Z 38} c_vel
LIN {X 75, Y 234, Z 38} c_vel
LIN {X 71, Y 240, Z 38} c_vel
LIN {X 66, Y 245, Z 38} c_vel
LIN {X 60, Y 250, Z 38} c_vel
LIN {X 52, Y 256, Z 38} c_vel
LIN {X 42, Y 261, Z 38} c_vel
LIN {X 30, Y 267, Z 38} c_vel
LIN {X 16, Y 273, Z 38} c_vel
LIN {X 0, Y 278, Z 38} c_vel
LIN {X 14, Y 327, Z 38} c_vel
LIN {X 28, Y 322, Z 38} c_vel
LIN {X 43, Y 317, Z 38} c_vel
LIN {X 57, Y 311, Z 38} c_vel
LIN {X 70, Y 304, Z 38} c_vel
LIN {X 81, Y 298, Z 38} c_vel
LIN {X 90, Y 291, Z 38} c_vel
LIN {X 99, Y 284, Z 38} c_vel
LIN {X 106, Y 277, Z 38} c_vel
LIN {X 113, Y 269, Z 38} c_vel
LIN {X 118, Y 261, Z 38} c_vel
LIN {X 123, Y 253, Z 38} c_vel
LIN {X 127, Y 244, Z 38} c_vel
LIN {X 130, Y 235, Z 38} c_vel
LIN {X 131, Y 226, Z 38} c_vel
LIN {X 133, Y 217, Z 38} c_vel
LIN {X 133, Y 207, Z 38} c_vel
LIN {X 133, Y 197, Z 38} c_vel
LIN {X 131, Y 186, Z 38} c_vel
LIN {X 129, Y 173, Z 38} c_vel
LIN {X 126, Y 160, Z 38} c_vel
LIN {X 120, Y 138, Z 38} c_vel
LIN {X 115, Y 118, Z 38} c_vel
LIN {X 112, Y 106, Z 38} c_vel
LIN {X 111, Y 96, Z 38} c_vel
LIN {X 110, Y 88, Z 38} c_vel
LIN {X 110, Y 81, Z 38} c_vel
LIN {X 111, Y 74, Z 38} c_vel
LIN {X 113, Y 69, Z 38} c_vel
LIN {X 116, Y 63, Z 38} c_vel
LIN {X 119, Y 58, Z 38} c_vel
LIN {X 124, Y 53, Z 38} c_vel
LIN {X 130, Y 48, Z 38} c_vel
LIN {X 138, Y 43, Z 38} c_vel
LIN {X 111, Y 0, Z 38} c_vel
$OUT[4] = FALSE
WAIT SEC 10.0
LIN {X 111, Y 0, Z 39} c_vel
$OUT[4] = TRUE
LIN {X 111, Y 0, Z 39} c_vel
LIN {X 106, Y 3, Z 39} c_vel
LIN {X 97, Y 9, Z 39} c_vel
LIN {X 89, Y 16, Z 39} c_vel
LIN {X 83, Y 23, Z 39} c_vel
LIN {X 77, Y 31, Z 39} c_vel
LIN {X 71, Y 39, Z 39} c_vel
LIN {X 67, Y 47, Z 39} c_vel
LIN {X 64, Y 56, Z 39} c_vel
LIN {X 62, Y 64, Z 39} c_vel
LIN {X 60, Y 73, Z 39} c_vel
LIN {X 59, Y 82, Z 39} c_vel
LIN {X 59, Y 92, Z 39} c_vel
LIN {X 60, Y 103, Z 39} c_vel
LIN {X 62, Y 114, Z 39} c_vel
LIN {X 65, Y 127, Z 39} c_vel
LIN {X 69, Y 144, Z 39} c_vel
LIN {X 74, Y 163, Z 39} c_vel
LIN {X 79, Y 180, Z 39} c_vel
LIN {X 81, Y 191, Z 39} c_vel
LIN {X 82, Y 201, Z 39} c_vel
LIN {X 82, Y 209, Z 39} c_vel
LIN {X 82, Y 217, Z 39} c_vel
LIN {X 80, Y 223, Z 39} c_vel
LIN {X 78, Y 229, Z 39} c_vel
LIN {X 75, Y 234, Z 39} c_vel
LIN {X 71, Y 240, Z 39} c_vel
LIN {X 66, Y 245, Z 39} c_vel
LIN {X 60, Y 250, Z 39} c_vel
LIN {X 52, Y 256, Z 39} c_vel
LIN {X 42, Y 261, Z 39} c_vel
LIN {X 30, Y 267, Z 39} c_vel
LIN {X 16, Y 273, Z 39} c_vel
LIN {X 0, Y 278, Z 39} c_vel
LIN {X 14, Y 327, Z 39} c_vel
LIN {X 28, Y 322, Z 39} c_vel
LIN {X 43, Y 317, Z 39} c_vel
LIN {X 57, Y 311, Z 39} c_vel
LIN {X 70, Y 304, Z 39} c_vel
LIN {X 81, Y 298, Z 39} c_vel
LIN {X 90, Y 291, Z 39} c_vel
LIN {X 99, Y 284, Z 39} c_vel
LIN {X 106, Y 277, Z 39} c_vel
LIN {X 113, Y 269, Z 39} c_vel
LIN {X 118, Y 261, Z 39} c_vel
LIN {X 123, Y 253, Z 39} c_vel
LIN {X 127, Y 244, Z 39} c_vel
LIN {X 130, Y 235, Z 39} c_vel
LIN {X 131, Y 226, Z 39} c_vel
LIN {X 133, Y 217, Z 39} c_vel
LIN {X 133, Y 207, Z 39} c_vel
LIN {X 133, Y 197, Z 39} c_vel
LIN {X 131, Y 186, Z 39} c_vel
LIN {X 129, Y 173, Z 39} c_vel
LIN {X 126, Y 160, Z 39} c_vel
LIN {X 120, Y 138, Z 39} c_vel
LIN {X 115, Y 118, Z 39} c_vel
LIN {X 112, Y 106, Z 39} c_vel
LIN {X 111, Y 96, Z 39} c_vel
LIN {X 110, Y 88, Z 39} c_vel
LIN {X 110, Y 81, Z 39} c_vel
LIN {X 111, Y 74, Z 39} c_vel
LIN {X 113, Y 69, Z 39} c_vel
LIN {X 116, Y 63, Z 39} c_vel
LIN {X 119, Y 58, Z 39} c_vel
LIN {X 124, Y 53, Z 39} c_vel
LIN {X 130, Y 48, Z 39} c_vel
LIN {X 138, Y 43, Z 39} c_vel
LIN {X 111, Y 0, Z 39} c_vel
$OUT[4] = FALSE
WAIT SEC 10.0
LIN {X 111, Y 0, Z 40} c_vel
$OUT[4] = TRUE
LIN {X 111, Y 0, Z 40} c_vel
LIN {X 106, Y 3, Z 40} c_vel
LIN {X 97, Y 9, Z 40} c_vel
LIN {X 89, Y 16, Z 40} c_vel
LIN {X 83, Y 23, Z 40} c_vel
LIN {X 77, Y 31, Z 40} c_vel
LIN {X 71, Y 39, Z 40} c_vel
LIN {X 67, Y 47, Z 40} c_vel
LIN {X 64, Y 56, Z 40} c_vel
LIN {X 62, Y 64, Z 40} c_vel
LIN {X 60, Y 73, Z 40} c_vel
LIN {X 59, Y 82, Z 40} c_vel
LIN {X 59, Y 92, Z 40} c_vel
LIN {X 60, Y 103, Z 40} c_vel
LIN {X 62, Y 114, Z 40} c_vel
LIN {X 65, Y 127, Z 40} c_vel
LIN {X 69, Y 144, Z 40} c_vel
LIN {X 74, Y 163, Z 40} c_vel
LIN {X 79, Y 180, Z 40} c_vel
LIN {X 81, Y 191, Z 40} c_vel
LIN {X 82, Y 201, Z 40} c_vel
LIN {X 82, Y 209, Z 40} c_vel
LIN {X 82, Y 217, Z 40} c_vel
LIN {X 80, Y 223, Z 40} c_vel
LIN {X 78, Y 229, Z 40} c_vel
LIN {X 75, Y 234, Z 40} c_vel
LIN {X 71, Y 240, Z 40} c_vel
LIN {X 66, Y 245, Z 40} c_vel
LIN {X 60, Y 250, Z 40} c_vel
LIN {X 52, Y 256, Z 40} c_vel
LIN {X 42, Y 261, Z 40} c_vel
LIN {X 30, Y 267, Z 40} c_vel
LIN {X 16, Y 273, Z 40} c_vel
LIN {X 0, Y 278, Z 40} c_vel
LIN {X 14, Y 327, Z 40} c_vel
LIN {X 28, Y 322, Z 40} c_vel
LIN {X 43, Y 317, Z 40} c_vel
LIN {X 57, Y 311, Z 40} c_vel
LIN {X 70, Y 304, Z 40} c_vel
LIN {X 81, Y 298, Z 40} c_vel
LIN {X 90, Y 291, Z 40} c_vel
LIN {X 99, Y 284, Z 40} c_vel
LIN {X 106, Y 277, Z 40} c_vel
LIN {X 113, Y 269, Z 40} c_vel
LIN {X 118, Y 261, Z 40} c_vel
LIN {X 123, Y 253, Z 40} c_vel
LIN {X 127, Y 244, Z 40} c_vel
LIN {X 130, Y 235, Z 40} c_vel
LIN {X 131, Y 226, Z 40} c_vel
LIN {X 133, Y 217, Z 40} c_vel
LIN {X 133, Y 207, Z 40} c_vel
LIN {X 133, Y 197, Z 40} c_vel
LIN {X 131, Y 186, Z 40} c_vel
LIN {X 129, Y 173, Z 40} c_vel
LIN {X 126, Y 160, Z 40} c_vel
LIN {X 120, Y 138, Z 40} c_vel
LIN {X 115, Y 118, Z 40} c_vel
LIN {X 112, Y 106, Z 40} c_vel
LIN {X 111, Y 96, Z 40} c_vel
LIN {X 110, Y 88, Z 40} c_vel
LIN {X 110, Y 81, Z 40} c_vel
LIN {X 111, Y 74, Z 40} c_vel
LIN {X 113, Y 69, Z 40} c_vel
LIN {X 116, Y 63, Z 40} c_vel
LIN {X 119, Y 58, Z 40} c_vel
LIN {X 124, Y 53, Z 40} c_vel
LIN {X 130, Y 48, Z 40} c_vel
LIN {X 138, Y 43, Z 40} c_vel
LIN {X 111, Y 0, Z 40} c_vel
$OUT[4] = FALSE
WAIT SEC 10.0
LIN {X 111, Y 0, Z 41} c_vel
$OUT[4] = TRUE
LIN {X 111, Y 0, Z 41} c_vel
LIN {X 106, Y 3, Z 41} c_vel
LIN {X 97, Y 9, Z 41} c_vel
LIN {X 89, Y 16, Z 41} c_vel
LIN {X 83, Y 23, Z 41} c_vel
LIN {X 77, Y 31, Z 41} c_vel
LIN {X 71, Y 39, Z 41} c_vel
LIN {X 67, Y 47, Z 41} c_vel
LIN {X 64, Y 56, Z 41} c_vel
LIN {X 62, Y 64, Z 41} c_vel
LIN {X 60, Y 73, Z 41} c_vel
LIN {X 59, Y 82, Z 41} c_vel
LIN {X 59, Y 92, Z 41} c_vel
LIN {X 60, Y 103, Z 41} c_vel
LIN {X 62, Y 114, Z 41} c_vel
LIN {X 65, Y 127, Z 41} c_vel
LIN {X 69, Y 144, Z 41} c_vel
LIN {X 74, Y 163, Z 41} c_vel
LIN {X 79, Y 180, Z 41} c_vel
LIN {X 81, Y 191, Z 41} c_vel
LIN {X 82, Y 201, Z 41} c_vel
LIN {X 82, Y 209, Z 41} c_vel
LIN {X 82, Y 217, Z 41} c_vel
LIN {X 80, Y 223, Z 41} c_vel
LIN {X 78, Y 229, Z 41} c_vel
LIN {X 75, Y 234, Z 41} c_vel
LIN {X 71, Y 240, Z 41} c_vel
LIN {X 66, Y 245, Z 41} c_vel
LIN {X 60, Y 250, Z 41} c_vel
LIN {X 52, Y 256, Z 41} c_vel
LIN {X 42, Y 261, Z 41} c_vel
LIN {X 30, Y 267, Z 41} c_vel
LIN {X 16, Y 273, Z 41} c_vel
LIN {X 0, Y 278, Z 41} c_vel
LIN {X 14, Y 327, Z 41} c_vel
LIN {X 28, Y 322, Z 41} c_vel
LIN {X 43, Y 317, Z 41} c_vel
LIN {X 57, Y 311, Z 41} c_vel
LIN {X 70, Y 304, Z 41} c_vel
LIN {X 81, Y 298, Z 41} c_vel
LIN {X 90, Y 291, Z 41} c_vel
LIN {X 99, Y 284, Z 41} c_vel
LIN {X 106, Y 277, Z 41} c_vel
LIN {X 113, Y 269, Z 41} c_vel
LIN {X 118, Y 261, Z 41} c_vel
LIN {X 123, Y 253, Z 41} c_vel
LIN {X 127, Y 244, Z 41} c_vel
LIN {X 130, Y 235, Z 41} c_vel
LIN {X 131, Y 226, Z 41} c_vel
LIN {X 133, Y 217, Z 41} c_vel
LIN {X 133, Y 207, Z 41} c_vel
LIN {X 133, Y 197, Z 41} c_vel
LIN {X 131, Y 186, Z 41} c_vel
LIN {X 129, Y 173, Z 41} c_vel
LIN {X 126, Y 160, Z 41} c_vel
LIN {X 120, Y 138, Z 41} c_vel
LIN {X 115, Y 118, Z 41} c_vel
LIN {X 112, Y 106, Z 41} c_vel
LIN {X 111, Y 96, Z 41} c_vel
LIN {X 110, Y 88, Z 41} c_vel
LIN {X 110, Y 81, Z 41} c_vel
LIN {X 111, Y 74, Z 41} c_vel
LIN {X 113, Y 69, Z 41} c_vel
LIN {X 116, Y 63, Z 41} c_vel
LIN {X 119, Y 58, Z 41} c_vel
LIN {X 124, Y 53, Z 41} c_vel
LIN {X 130, Y 48, Z 41} c_vel
LIN {X 138, Y 43, Z 41} c_vel
LIN {X 111, Y 0, Z 41} c_vel
$OUT[4] = FALSE
WAIT SEC 10.0
LIN {X 111, Y 0, Z 42} c_vel
$OUT[4] = TRUE
LIN {X 111, Y 0, Z 42} c_vel
LIN {X 106, Y 3, Z 42} c_vel
LIN {X 97, Y 9, Z 42} c_vel
LIN {X 89, Y 16, Z 42} c_vel
LIN {X 83, Y 23, Z 42} c_vel
LIN {X 77, Y 31, Z 42} c_vel
LIN {X 71, Y 39, Z 42} c_vel
LIN {X 67, Y 47, Z 42} c_vel
LIN {X 64, Y 56, Z 42} c_vel
LIN {X 62, Y 64, Z 42} c_vel
LIN {X 60, Y 73, Z 42} c_vel
LIN {X 59, Y 82, Z 42} c_vel
LIN {X 59, Y 92, Z 42} c_vel
LIN {X 60, Y 103, Z 42} c_vel
LIN {X 62, Y 114, Z 42} c_vel
LIN {X 65, Y 127, Z 42} c_vel
LIN {X 69, Y 144, Z 42} c_vel
LIN {X 74, Y 163, Z 42} c_vel
LIN {X 79, Y 180, Z 42} c_vel
LIN {X 81, Y 191, Z 42} c_vel
LIN {X 82, Y 201, Z 42} c_vel
LIN {X 82, Y 209, Z 42} c_vel
LIN {X 82, Y 217, Z 42} c_vel
LIN {X 80, Y 223, Z 42} c_vel
LIN {X 78, Y 229, Z 42} c_vel
LIN {X 75, Y 234, Z 42} c_vel
LIN {X 71, Y 240, Z 42} c_vel
LIN {X 66, Y 245, Z 42} c_vel
LIN {X 60, Y 250, Z 42} c_vel
LIN {X 52, Y 256, Z 42} c_vel
LIN {X 42, Y 261, Z 42} c_vel
LIN {X 30, Y 267, Z 42} c_vel
LIN {X 16, Y 273, Z 42} c_vel
LIN {X 0, Y 278, Z 42} c_vel
LIN {X 14, Y 327, Z 42} c_vel
LIN {X 28, Y 322, Z 42} c_vel
LIN {X 43, Y 317, Z 42} c_vel
LIN {X 57, Y 311, Z 42} c_vel
LIN {X 70, Y 304, Z 42} c_vel
LIN {X 81, Y 298, Z 42} c_vel
LIN {X 90, Y 291, Z 42} c_vel
LIN {X 99, Y 284, Z 42} c_vel
LIN {X 106, Y 277, Z 42} c_vel
LIN {X 113, Y 269, Z 42} c_vel
LIN {X 118, Y 261, Z 42} c_vel
LIN {X 123, Y 253, Z 42} c_vel
LIN {X 127, Y 244, Z 42} c_vel
LIN {X 130, Y 235, Z 42} c_vel
LIN {X 131, Y 226, Z 42} c_vel
LIN {X 133, Y 217, Z 42} c_vel
LIN {X 133, Y 207, Z 42} c_vel
LIN {X 133, Y 197, Z 42} c_vel
LIN {X 131, Y 186, Z 42} c_vel
LIN {X 129, Y 173, Z 42} c_vel
LIN {X 126, Y 160, Z 42} c_vel
LIN {X 120, Y 138, Z 42} c_vel
LIN {X 115, Y 118, Z 42} c_vel
LIN {X 112, Y 106, Z 42} c_vel
LIN {X 111, Y 96, Z 42} c_vel
LIN {X 110, Y 88, Z 42} c_vel
LIN {X 110, Y 81, Z 42} c_vel
LIN {X 111, Y 74, Z 42} c_vel
LIN {X 113, Y 69, Z 42} c_vel
LIN {X 116, Y 63, Z 42} c_vel
LIN {X 119, Y 58, Z 42} c_vel
LIN {X 124, Y 53, Z 42} c_vel
LIN {X 130, Y 48, Z 42} c_vel
LIN {X 138, Y 43, Z 42} c_vel
LIN {X 111, Y 0, Z 42} c_vel
$OUT[4] = FALSE
WAIT SEC 10.0
LIN {X 111, Y 0, Z 43} c_vel
$OUT[4] = TRUE
LIN {X 111, Y 0, Z 43} c_vel
LIN {X 106, Y 3, Z 43} c_vel
LIN {X 97, Y 9, Z 43} c_vel
LIN {X 89, Y 16, Z 43} c_vel
LIN {X 83, Y 23, Z 43} c_vel
LIN {X 77, Y 31, Z 43} c_vel
LIN {X 71, Y 39, Z 43} c_vel
LIN {X 67, Y 47, Z 43} c_vel
LIN {X 64, Y 56, Z 43} c_vel
LIN {X 62, Y 64, Z 43} c_vel
LIN {X 60, Y 73, Z 43} c_vel
LIN {X 59, Y 82, Z 43} c_vel
LIN {X 59, Y 92, Z 43} c_vel
LIN {X 60, Y 103, Z 43} c_vel
LIN {X 62, Y 114, Z 43} c_vel
LIN {X 65, Y 127, Z 43} c_vel
LIN {X 69, Y 144, Z 43} c_vel
LIN {X 74, Y 163, Z 43} c_vel
LIN {X 79, Y 180, Z 43} c_vel
LIN {X 81, Y 191, Z 43} c_vel
LIN {X 82, Y 201, Z 43} c_vel
LIN {X 82, Y 209, Z 43} c_vel
LIN {X 82, Y 217, Z 43} c_vel
LIN {X 80, Y 223, Z 43} c_vel
LIN {X 78, Y 229, Z 43} c_vel
LIN {X 75, Y 234, Z 43} c_vel
LIN {X 71, Y 240, Z 43} c_vel
LIN {X 66, Y 245, Z 43} c_vel
LIN {X 60, Y 250, Z 43} c_vel
LIN {X 52, Y 256, Z 43} c_vel
LIN {X 42, Y 261, Z 43} c_vel
LIN {X 30, Y 267, Z 43} c_vel
LIN {X 16, Y 273, Z 43} c_vel
LIN {X 0, Y 278, Z 43} c_vel
LIN {X 14, Y 327, Z 43} c_vel
LIN {X 28, Y 322, Z 43} c_vel
LIN {X 43, Y 317, Z 43} c_vel
LIN {X 57, Y 311, Z 43} c_vel
LIN {X 70, Y 304, Z 43} c_vel
LIN {X 81, Y 298, Z 43} c_vel
LIN {X 90, Y 291, Z 43} c_vel
LIN {X 99, Y 284, Z 43} c_vel
LIN {X 106, Y 277, Z 43} c_vel
LIN {X 113, Y 269, Z 43} c_vel
LIN {X 118, Y 261, Z 43} c_vel
LIN {X 123, Y 253, Z 43} c_vel
LIN {X 127, Y 244, Z 43} c_vel
LIN {X 130, Y 235, Z 43} c_vel
LIN {X 131, Y 226, Z 43} c_vel
LIN {X 133, Y 217, Z 43} c_vel
LIN {X 133, Y 207, Z 43} c_vel
LIN {X 133, Y 197, Z 43} c_vel
LIN {X 131, Y 186, Z 43} c_vel
LIN {X 129, Y 173, Z 43} c_vel
LIN {X 126, Y 160, Z 43} c_vel
LIN {X 120, Y 138, Z 43} c_vel
LIN {X 115, Y 118, Z 43} c_vel
LIN {X 112, Y 106, Z 43} c_vel
LIN {X 111, Y 96, Z 43} c_vel
LIN {X 110, Y 88, Z 43} c_vel
LIN {X 110, Y 81, Z 43} c_vel
LIN {X 111, Y 74, Z 43} c_vel
LIN {X 113, Y 69, Z 43} c_vel
LIN {X 116, Y 63, Z 43} c_vel
LIN {X 119, Y 58, Z 43} c_vel
LIN {X 124, Y 53, Z 43} c_vel
LIN {X 130, Y 48, Z 43} c_vel
LIN {X 138, Y 43, Z 43} c_vel
LIN {X 111, Y 0, Z 43} c_vel
$OUT[4] = FALSE
WAIT SEC 10.0
LIN {X 111, Y 0, Z 44} c_vel
$OUT[4] = TRUE
LIN {X 111, Y 0, Z 44} c_vel
LIN {X 106, Y 3, Z 44} c_vel
LIN {X 97, Y 9, Z 44} c_vel
LIN {X 89, Y 16, Z 44} c_vel
LIN {X 83, Y 23, Z 44} c_vel
LIN {X 77, Y 31, Z 44} c_vel
LIN {X 71, Y 39, Z 44} c_vel
LIN {X 67, Y 47, Z 44} c_vel
LIN {X 64, Y 56, Z 44} c_vel
LIN {X 62, Y 64, Z 44} c_vel
LIN {X 60, Y 73, Z 44} c_vel
LIN {X 59, Y 82, Z 44} c_vel
LIN {X 59, Y 92, Z 44} c_vel
LIN {X 60, Y 103, Z 44} c_vel
LIN {X 62, Y 114, Z 44} c_vel
LIN {X 65, Y 127, Z 44} c_vel
LIN {X 69, Y 144, Z 44} c_vel
LIN {X 74, Y 163, Z 44} c_vel
LIN {X 79, Y 180, Z 44} c_vel
LIN {X 81, Y 191, Z 44} c_vel
LIN {X 82, Y 201, Z 44} c_vel
LIN {X 82, Y 209, Z 44} c_vel
LIN {X 82, Y 217, Z 44} c_vel
LIN {X 80, Y 223, Z 44} c_vel
LIN {X 78, Y 229, Z 44} c_vel
LIN {X 75, Y 234, Z 44} c_vel
LIN {X 71, Y 240, Z 44} c_vel
LIN {X 66, Y 245, Z 44} c_vel
LIN {X 60, Y 250, Z 44} c_vel
LIN {X 52, Y 256, Z 44} c_vel
LIN {X 42, Y 261, Z 44} c_vel
LIN {X 30, Y 267, Z 44} c_vel
LIN {X 16, Y 273, Z 44} c_vel
LIN {X 0, Y 278, Z 44} c_vel
LIN {X 14, Y 327, Z 44} c_vel
LIN {X 28, Y 322, Z 44} c_vel
LIN {X 43, Y 317, Z 44} c_vel
LIN {X 57, Y 311, Z 44} c_vel
LIN {X 70, Y 304, Z 44} c_vel
LIN {X 81, Y 298, Z 44} c_vel
LIN {X 90, Y 291, Z 44} c_vel
LIN {X 99, Y 284, Z 44} c_vel
LIN {X 106, Y 277, Z 44} c_vel
LIN {X 113, Y 269, Z 44} c_vel
LIN {X 118, Y 261, Z 44} c_vel
LIN {X 123, Y 253, Z 44} c_vel
LIN {X 127, Y 244, Z 44} c_vel
LIN {X 130, Y 235, Z 44} c_vel
LIN {X 131, Y 226, Z 44} c_vel
LIN {X 133, Y 217, Z 44} c_vel
LIN {X 133, Y 207, Z 44} c_vel
LIN {X 133, Y 197, Z 44} c_vel
LIN {X 131, Y 186, Z 44} c_vel
LIN {X 129, Y 173, Z 44} c_vel
LIN {X 126, Y 160, Z 44} c_vel
LIN {X 120, Y 138, Z 44} c_vel
LIN {X 115, Y 118, Z 44} c_vel
LIN {X 112, Y 106, Z 44} c_vel
LIN {X 111, Y 96, Z 44} c_vel
LIN {X 110, Y 88, Z 44} c_vel
LIN {X 110, Y 81, Z 44} c_vel
LIN {X 111, Y 74, Z 44} c_vel
LIN {X 113, Y 69, Z 44} c_vel
LIN {X 116, Y 63, Z 44} c_vel
LIN {X 119, Y 58, Z 44} c_vel
LIN {X 124, Y 53, Z 44} c_vel
LIN {X 130, Y 48, Z 44} c_vel
LIN {X 138, Y 43, Z 44} c_vel
LIN {X 111, Y 0, Z 44} c_vel
$OUT[4] = FALSE
WAIT SEC 10.0
LIN {X 111, Y 0, Z 45} c_vel
$OUT[4] = TRUE
LIN {X 111, Y 0, Z 45} c_vel
LIN {X 106, Y 3, Z 45} c_vel
LIN {X 97, Y 9, Z 45} c_vel
LIN {X 89, Y 16, Z 45} c_vel
LIN {X 83, Y 23, Z 45} c_vel
LIN {X 77, Y 31, Z 45} c_vel
LIN {X 71, Y 39, Z 45} c_vel
LIN {X 67, Y 47, Z 45} c_vel
LIN {X 64, Y 56, Z 45} c_vel
LIN {X 62, Y 64, Z 45} c_vel
LIN {X 60, Y 73, Z 45} c_vel
LIN {X 59, Y 82, Z 45} c_vel
LIN {X 59, Y 92, Z 45} c_vel
LIN {X 60, Y 103, Z 45} c_vel
LIN {X 62, Y 114, Z 45} c_vel
LIN {X 65, Y 127, Z 45} c_vel
LIN {X 69, Y 144, Z 45} c_vel
LIN {X 74, Y 163, Z 45} c_vel
LIN {X 79, Y 180, Z 45} c_vel
LIN {X 81, Y 191, Z 45} c_vel
LIN {X 82, Y 201, Z 45} c_vel
LIN {X 82, Y 209, Z 45} c_vel
LIN {X 82, Y 217, Z 45} c_vel
LIN {X 80, Y 223, Z 45} c_vel
LIN {X 78, Y 229, Z 45} c_vel
LIN {X 75, Y 234, Z 45} c_vel
LIN {X 71, Y 240, Z 45} c_vel
LIN {X 66, Y 245, Z 45} c_vel
LIN {X 60, Y 250, Z 45} c_vel
LIN {X 52, Y 256, Z 45} c_vel
LIN {X 42, Y 261, Z 45} c_vel
LIN {X 30, Y 267, Z 45} c_vel
LIN {X 16, Y 273, Z 45} c_vel
LIN {X 0, Y 278, Z 45} c_vel
LIN {X 14, Y 327, Z 45} c_vel
LIN {X 28, Y 322, Z 45} c_vel
LIN {X 43, Y 317, Z 45} c_vel
LIN {X 57, Y 311, Z 45} c_vel
LIN {X 70, Y 304, Z 45} c_vel
LIN {X 81, Y 298, Z 45} c_vel
LIN {X 90, Y 291, Z 45} c_vel
LIN {X 99, Y 284, Z 45} c_vel
LIN {X 106, Y 277, Z 45} c_vel
LIN {X 113, Y 269, Z 45} c_vel
LIN {X 118, Y 261, Z 45} c_vel
LIN {X 123, Y 253, Z 45} c_vel
LIN {X 127, Y 244, Z 45} c_vel
LIN {X 130, Y 235, Z 45} c_vel
LIN {X 131, Y 226, Z 45} c_vel
LIN {X 133, Y 217, Z 45} c_vel
LIN {X 133, Y 207, Z 45} c_vel
LIN {X 133, Y 197, Z 45} c_vel
LIN {X 131, Y 186, Z 45} c_vel
LIN {X 129, Y 173, Z 45} c_vel
LIN {X 126, Y 160, Z 45} c_vel
LIN {X 120, Y 138, Z 45} c_vel
LIN {X 115, Y 118, Z 45} c_vel
LIN {X 112, Y 106, Z 45} c_vel
LIN {X 111, Y 96, Z 45} c_vel
LIN {X 110, Y 88, Z 45} c_vel
LIN {X 110, Y 81, Z 45} c_vel
LIN {X 111, Y 74, Z 45} c_vel
LIN {X 113, Y 69, Z 45} c_vel
LIN {X 116, Y 63, Z 45} c_vel
LIN {X 119, Y 58, Z 45} c_vel
LIN {X 124, Y 53, Z 45} c_vel
LIN {X 130, Y 48, Z 45} c_vel
LIN {X 138, Y 43, Z 45} c_vel
LIN {X 111, Y 0, Z 45} c_vel
$OUT[4] = FALSE
WAIT SEC 10.0
LIN {X 111, Y 0, Z 46} c_vel
$OUT[4] = TRUE
LIN {X 111, Y 0, Z 46} c_vel
LIN {X 106, Y 3, Z 46} c_vel
LIN {X 97, Y 9, Z 46} c_vel
LIN {X 89, Y 16, Z 46} c_vel
LIN {X 83, Y 23, Z 46} c_vel
LIN {X 77, Y 31, Z 46} c_vel
LIN {X 71, Y 39, Z 46} c_vel
LIN {X 67, Y 47, Z 46} c_vel
LIN {X 64, Y 56, Z 46} c_vel
LIN {X 62, Y 64, Z 46} c_vel
LIN {X 60, Y 73, Z 46} c_vel
LIN {X 59, Y 82, Z 46} c_vel
LIN {X 59, Y 92, Z 46} c_vel
LIN {X 60, Y 103, Z 46} c_vel
LIN {X 62, Y 114, Z 46} c_vel
LIN {X 65, Y 127, Z 46} c_vel
LIN {X 69, Y 144, Z 46} c_vel
LIN {X 74, Y 163, Z 46} c_vel
LIN {X 79, Y 180, Z 46} c_vel
LIN {X 81, Y 191, Z 46} c_vel
LIN {X 82, Y 201, Z 46} c_vel
LIN {X 82, Y 209, Z 46} c_vel
LIN {X 82, Y 217, Z 46} c_vel
LIN {X 80, Y 223, Z 46} c_vel
LIN {X 78, Y 229, Z 46} c_vel
LIN {X 75, Y 234, Z 46} c_vel
LIN {X 71, Y 240, Z 46} c_vel
LIN {X 66, Y 245, Z 46} c_vel
LIN {X 60, Y 250, Z 46} c_vel
LIN {X 52, Y 256, Z 46} c_vel
LIN {X 42, Y 261, Z 46} c_vel
LIN {X 30, Y 267, Z 46} c_vel
LIN {X 16, Y 273, Z 46} c_vel
LIN {X 0, Y 278, Z 46} c_vel
LIN {X 14, Y 327, Z 46} c_vel
LIN {X 28, Y 322, Z 46} c_vel
LIN {X 43, Y 317, Z 46} c_vel
LIN {X 57, Y 311, Z 46} c_vel
LIN {X 70, Y 304, Z 46} c_vel
LIN {X 81, Y 298, Z 46} c_vel
LIN {X 90, Y 291, Z 46} c_vel
LIN {X 99, Y 284, Z 46} c_vel
LIN {X 106, Y 277, Z 46} c_vel
LIN {X 113, Y 269, Z 46} c_vel
LIN {X 118, Y 261, Z 46} c_vel
LIN {X 123, Y 253, Z 46} c_vel
LIN {X 127, Y 244, Z 46} c_vel
LIN {X 130, Y 235, Z 46} c_vel
LIN {X 131, Y 226, Z 46} c_vel
LIN {X 133, Y 217, Z 46} c_vel
LIN {X 133, Y 207, Z 46} c_vel
LIN {X 133, Y 197, Z 46} c_vel
LIN {X 131, Y 186, Z 46} c_vel
LIN {X 129, Y 173, Z 46} c_vel
LIN {X 126, Y 160, Z 46} c_vel
LIN {X 120, Y 138, Z 46} c_vel
LIN {X 115, Y 118, Z 46} c_vel
LIN {X 112, Y 106, Z 46} c_vel
LIN {X 111, Y 96, Z 46} c_vel
LIN {X 110, Y 88, Z 46} c_vel
LIN {X 110, Y 81, Z 46} c_vel
LIN {X 111, Y 74, Z 46} c_vel
LIN {X 113, Y 69, Z 46} c_vel
LIN {X 116, Y 63, Z 46} c_vel
LIN {X 119, Y 58, Z 46} c_vel
LIN {X 124, Y 53, Z 46} c_vel
LIN {X 130, Y 48, Z 46} c_vel
LIN {X 138, Y 43, Z 46} c_vel
LIN {X 111, Y 0, Z 46} c_vel
$OUT[4] = FALSE
WAIT SEC 10.0
LIN {X 111, Y 0, Z 47} c_vel
$OUT[4] = TRUE
LIN {X 111, Y 0, Z 47} c_vel
LIN {X 106, Y 3, Z 47} c_vel
LIN {X 97, Y 9, Z 47} c_vel
LIN {X 89, Y 16, Z 47} c_vel
LIN {X 83, Y 23, Z 47} c_vel
LIN {X 77, Y 31, Z 47} c_vel
LIN {X 71, Y 39, Z 47} c_vel
LIN {X 67, Y 47, Z 47} c_vel
LIN {X 64, Y 56, Z 47} c_vel
LIN {X 62, Y 64, Z 47} c_vel
LIN {X 60, Y 73, Z 47} c_vel
LIN {X 59, Y 82, Z 47} c_vel
LIN {X 59, Y 92, Z 47} c_vel
LIN {X 60, Y 103, Z 47} c_vel
LIN {X 62, Y 114, Z 47} c_vel
LIN {X 65, Y 127, Z 47} c_vel
LIN {X 69, Y 144, Z 47} c_vel
LIN {X 74, Y 163, Z 47} c_vel
LIN {X 79, Y 180, Z 47} c_vel
LIN {X 81, Y 191, Z 47} c_vel
LIN {X 82, Y 201, Z 47} c_vel
LIN {X 82, Y 209, Z 47} c_vel
LIN {X 82, Y 217, Z 47} c_vel
LIN {X 80, Y 223, Z 47} c_vel
LIN {X 78, Y 229, Z 47} c_vel
LIN {X 75, Y 234, Z 47} c_vel
LIN {X 71, Y 240, Z 47} c_vel
LIN {X 66, Y 245, Z 47} c_vel
LIN {X 60, Y 250, Z 47} c_vel
